REGION Network 63: Reset CMS
   // Reset Axis when the unit is in the resetting state.
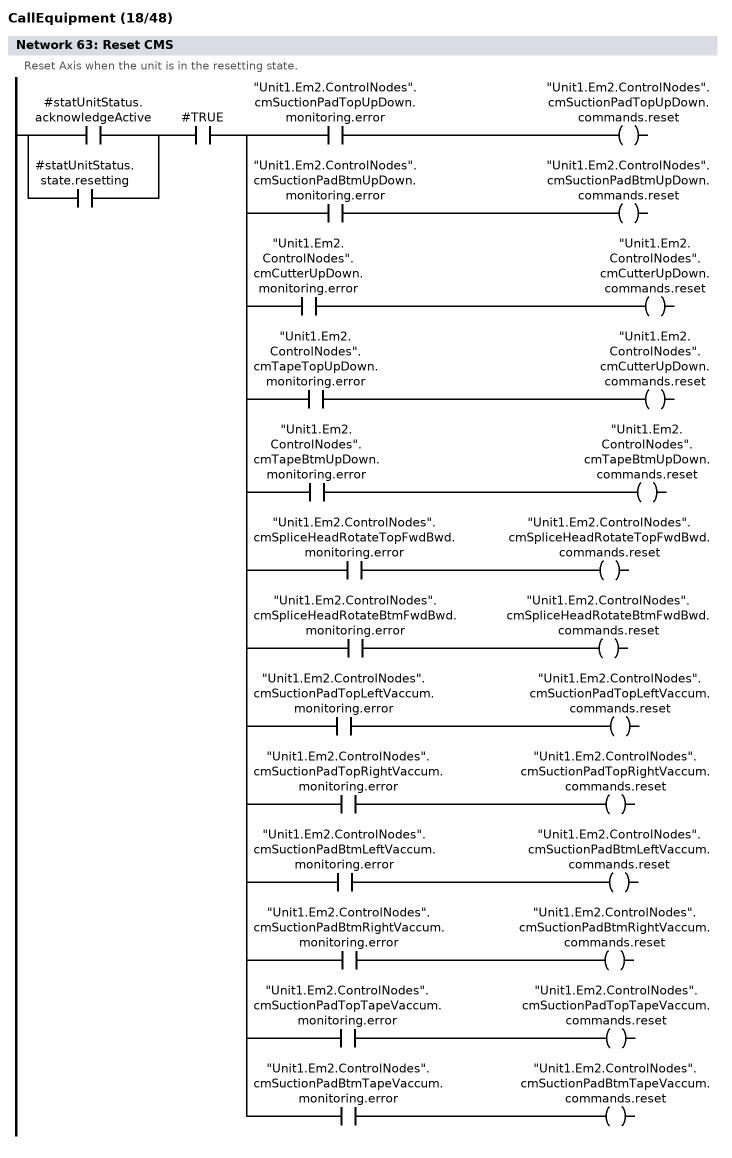
   RUNG wire#powerrail
      Contact( #statUnitStatus.acknowledgeActive )
      wire#w1
      Contact( #TRUE )
      wire#w2
      Contact( "Unit1.Em2.ControlNodes".cmSuctionPadTopUpDown.monitoring.error )
      Coil( "Unit1.Em2.ControlNodes".cmSuctionPadTopUpDown.commands.reset )
   END_RUNG
   RUNG wire#powerrail
      Contact( #statUnitStatus.state.resetting )
   END_RUNG wire#w1
   RUNG wire#w2
      Contact( "Unit1.Em2.ControlNodes".cmSuctionPadBtmUpDown.monitoring.error )
      Coil( "Unit1.Em2.ControlNodes".cmSuctionPadBtmUpDown.commands.reset )
   END_RUNG
   RUNG wire#w2
      Contact( "Unit1.Em2.ControlNodes".cmCutterUpDown.monitoring.error )
      Coil( "Unit1.Em2.ControlNodes".cmCutterUpDown.commands.reset )
   END_RUNG
   RUNG wire#w2
      Contact( "Unit1.Em2.ControlNodes".cmTapeTopUpDown.monitoring.error )
      Coil( "Unit1.Em2.ControlNodes".cmCutterUpDown.commands.reset )
   END_RUNG
   RUNG wire#w2
      Contact( "Unit1.Em2.ControlNodes".cmTapeBtmUpDown.monitoring.error )
      Coil( "Unit1.Em2.ControlNodes".cmTapeBtmUpDown.commands.reset )
   END_RUNG
   RUNG wire#w2
      Contact( "Unit1.Em2.ControlNodes".cmSpliceHeadRotateTopFwdBwd.monitoring.error )
      Coil( "Unit1.Em2.ControlNodes".cmSpliceHeadRotateTopFwdBwd.commands.reset )
   END_RUNG
   RUNG wire#w2
      Contact( "Unit1.Em2.ControlNodes".cmSpliceHeadRotateBtmFwdBwd.monitoring.error )
      Coil( "Unit1.Em2.ControlNodes".cmSpliceHeadRotateBtmFwdBwd.commands.reset )
   END_RUNG
   RUNG wire#w2
      Contact( "Unit1.Em2.ControlNodes".cmSuctionPadTopLeftVaccum.monitoring.error )
      Coil( "Unit1.Em2.ControlNodes".cmSuctionPadTopLeftVaccum.commands.reset )
   END_RUNG
   RUNG wire#w2
      Contact( "Unit1.Em2.ControlNodes".cmSuctionPadTopRightVaccum.monitoring.error )
      Coil( "Unit1.Em2.ControlNodes".cmSuctionPadTopRightVaccum.commands.reset )
   END_RUNG
   RUNG wire#w2
      Contact( "Unit1.Em2.ControlNodes".cmSuctionPadBtmLeftVaccum.monitoring.error )
      Coil( "Unit1.Em2.ControlNodes".cmSuctionPadBtmLeftVaccum.commands.reset )
   END_RUNG
   RUNG wire#w2
      Contact( "Unit1.Em2.ControlNodes".cmSuctionPadBtmRightVaccum.monitoring.error )
      Coil( "Unit1.Em2.ControlNodes".cmSuctionPadBtmRightVaccum.commands.reset )
   END_RUNG
   RUNG wire#w2
      Contact( "Unit1.Em2.ControlNodes".cmSuctionPadTopTapeVaccum.monitoring.error )
      Coil( "Unit1.Em2.ControlNodes".cmSuctionPadTopTapeVaccum.commands.reset )
   END_RUNG
   RUNG wire#w2
      Contact( "Unit1.Em2.ControlNodes".cmSuctionPadBtmTapeVaccum.monitoring.error )
      Coil( "Unit1.Em2.ControlNodes".cmSuctionPadBtmTapeVaccum.commands.reset )
   END_RUNG
   // the same network as SCL:
   #_w1 := (#statUnitStatus.acknowledgeActive OR #statUnitStatus.state.resetting) AND #TRUE;
   "Unit1.Em2.ControlNodes".cmSuctionPadTopUpDown.commands.reset := #_w1 AND "Unit1.Em2.ControlNodes".cmSuctionPadTopUpDown.monitoring.error;
   "Unit1.Em2.ControlNodes".cmSuctionPadBtmUpDown.commands.reset := #_w1 AND "Unit1.Em2.ControlNodes".cmSuctionPadBtmUpDown.monitoring.error;
   "Unit1.Em2.ControlNodes".cmCutterUpDown.commands.reset := #_w1 AND "Unit1.Em2.ControlNodes".cmCutterUpDown.monitoring.error;
   "Unit1.Em2.ControlNodes".cmCutterUpDown.commands.reset := #_w1 AND "Unit1.Em2.ControlNodes".cmTapeTopUpDown.monitoring.error;
   "Unit1.Em2.ControlNodes".cmTapeBtmUpDown.commands.reset := #_w1 AND "Unit1.Em2.ControlNodes".cmTapeBtmUpDown.monitoring.error;
   "Unit1.Em2.ControlNodes".cmSpliceHeadRotateTopFwdBwd.commands.reset := #_w1 AND "Unit1.Em2.ControlNodes".cmSpliceHeadRotateTopFwdBwd.monitoring.error;
   "Unit1.Em2.ControlNodes".cmSpliceHeadRotateBtmFwdBwd.commands.reset := #_w1 AND "Unit1.Em2.ControlNodes".cmSpliceHeadRotateBtmFwdBwd.monitoring.error;
   "Unit1.Em2.ControlNodes".cmSuctionPadTopLeftVaccum.commands.reset := #_w1 AND "Unit1.Em2.ControlNodes".cmSuctionPadTopLeftVaccum.monitoring.error;
   "Unit1.Em2.ControlNodes".cmSuctionPadTopRightVaccum.commands.reset := #_w1 AND "Unit1.Em2.ControlNodes".cmSuctionPadTopRightVaccum.monitoring.error;
   "Unit1.Em2.ControlNodes".cmSuctionPadBtmLeftVaccum.commands.reset := #_w1 AND "Unit1.Em2.ControlNodes".cmSuctionPadBtmLeftVaccum.monitoring.error;
   "Unit1.Em2.ControlNodes".cmSuctionPadBtmRightVaccum.commands.reset := #_w1 AND "Unit1.Em2.ControlNodes".cmSuctionPadBtmRightVaccum.monitoring.error;
   "Unit1.Em2.ControlNodes".cmSuctionPadTopTapeVaccum.commands.reset := #_w1 AND "Unit1.Em2.ControlNodes".cmSuctionPadTopTapeVaccum.monitoring.error;
   "Unit1.Em2.ControlNodes".cmSuctionPadBtmTapeVaccum.commands.reset := #_w1 AND "Unit1.Em2.ControlNodes".cmSuctionPadBtmTapeVaccum.monitoring.error;
END_REGION

REGION Network 65: cmSuctionPadTopUpDown Interlock
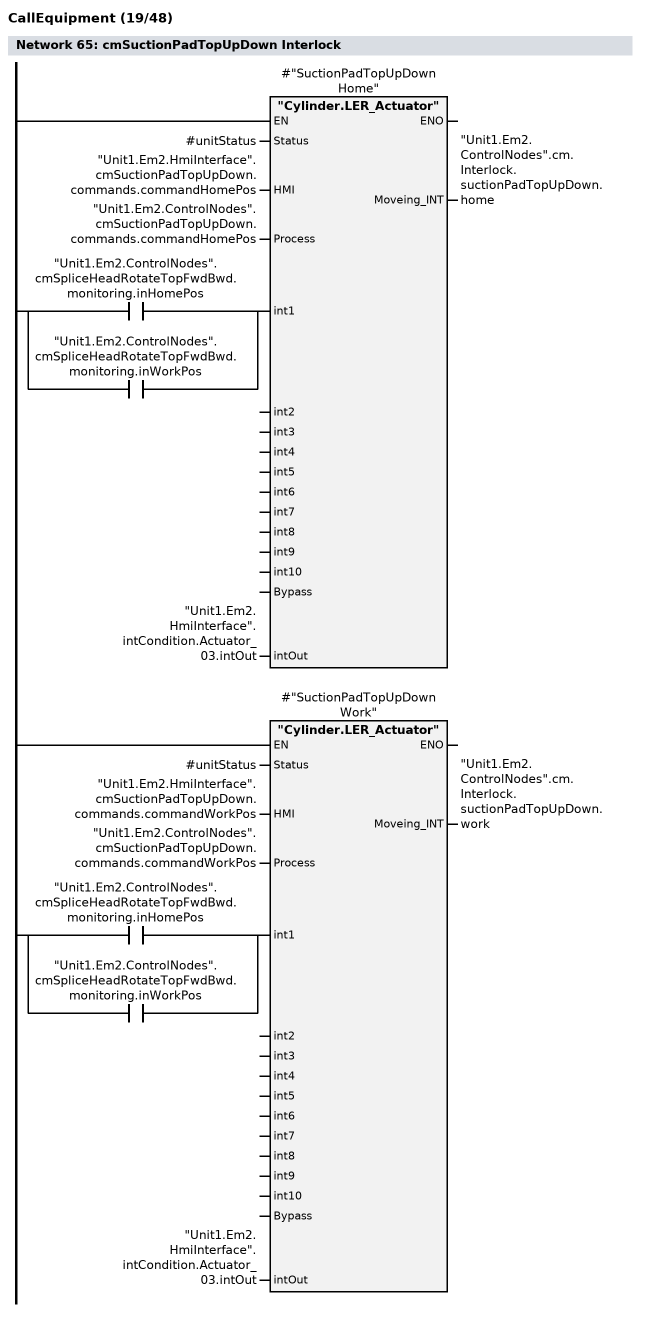
   RUNG wire#powerrail
      #"SuctionPadTopUpDown Home"(int1 := wire#w1, Status := #unitStatus, HMI := "Unit1.Em2.HmiInterface".cmSuctionPadTopUpDown.commands.commandHomePos, Process := "Unit1.Em2.ControlNodes".cmSuctionPadTopUpDown.commands.commandHomePos, int2 :=, int3 :=, int4 :=, int5 :=, int6 :=, int7 :=, int8 :=, int9 :=, int10 :=, Bypass :=, intOut := "Unit1.Em2.HmiInterface".intCondition.Actuator_03.intOut, Moveing_INT => "Unit1.Em2.ControlNodes".cm.Interlock.suctionPadTopUpDown.home)
   END_RUNG
   RUNG wire#powerrail
      Contact( "Unit1.Em2.ControlNodes".cmSpliceHeadRotateTopFwdBwd.monitoring.inHomePos )
   END_RUNG wire#w1
   RUNG wire#powerrail
      Contact( "Unit1.Em2.ControlNodes".cmSpliceHeadRotateTopFwdBwd.monitoring.inWorkPos )
   END_RUNG wire#w1
   RUNG wire#powerrail
      #"SuctionPadTopUpDown Work"(int1 := wire#w2, Status := #unitStatus, HMI := "Unit1.Em2.HmiInterface".cmSuctionPadTopUpDown.commands.commandWorkPos, Process := "Unit1.Em2.ControlNodes".cmSuctionPadTopUpDown.commands.commandWorkPos, int2 :=, int3 :=, int4 :=, int5 :=, int6 :=, int7 :=, int8 :=, int9 :=, int10 :=, Bypass :=, intOut := "Unit1.Em2.HmiInterface".intCondition.Actuator_03.intOut, Moveing_INT => "Unit1.Em2.ControlNodes".cm.Interlock.suctionPadTopUpDown.work)
   END_RUNG
   RUNG wire#powerrail
      Contact( "Unit1.Em2.ControlNodes".cmSpliceHeadRotateTopFwdBwd.monitoring.inHomePos )
   END_RUNG wire#w2
   RUNG wire#powerrail
      Contact( "Unit1.Em2.ControlNodes".cmSpliceHeadRotateTopFwdBwd.monitoring.inWorkPos )
   END_RUNG wire#w2
   // the same network as SCL:
   #"SuctionPadTopUpDown Home"(Status := #unitStatus,   // "Cylinder.LER_Actuator"
                           HMI := "Unit1.Em2.HmiInterface".cmSuctionPadTopUpDown.commands.commandHomePos,
                           Process := "Unit1.Em2.ControlNodes".cmSuctionPadTopUpDown.commands.commandHomePos,
                           int1 := "Unit1.Em2.ControlNodes".cmSpliceHeadRotateTopFwdBwd.monitoring.inHomePos OR "Unit1.Em2.ControlNodes".cmSpliceHeadRotateTopFwdBwd.monitoring.inWorkPos,
                           intOut := "Unit1.Em2.HmiInterface".intCondition.Actuator_03.intOut,
                           Moveing_INT => "Unit1.Em2.ControlNodes".cm.Interlock.suctionPadTopUpDown.home);
   #"SuctionPadTopUpDown Work"(Status := #unitStatus,   // "Cylinder.LER_Actuator"
                           HMI := "Unit1.Em2.HmiInterface".cmSuctionPadTopUpDown.commands.commandWorkPos,
                           Process := "Unit1.Em2.ControlNodes".cmSuctionPadTopUpDown.commands.commandWorkPos,
                           int1 := "Unit1.Em2.ControlNodes".cmSpliceHeadRotateTopFwdBwd.monitoring.inHomePos OR "Unit1.Em2.ControlNodes".cmSpliceHeadRotateTopFwdBwd.monitoring.inWorkPos,
                           intOut := "Unit1.Em2.HmiInterface".intCondition.Actuator_03.intOut,
                           Moveing_INT => "Unit1.Em2.ControlNodes".cm.Interlock.suctionPadTopUpDown.work);
END_REGION

REGION Network 66: cmSuctionPadTopUpDown Commands
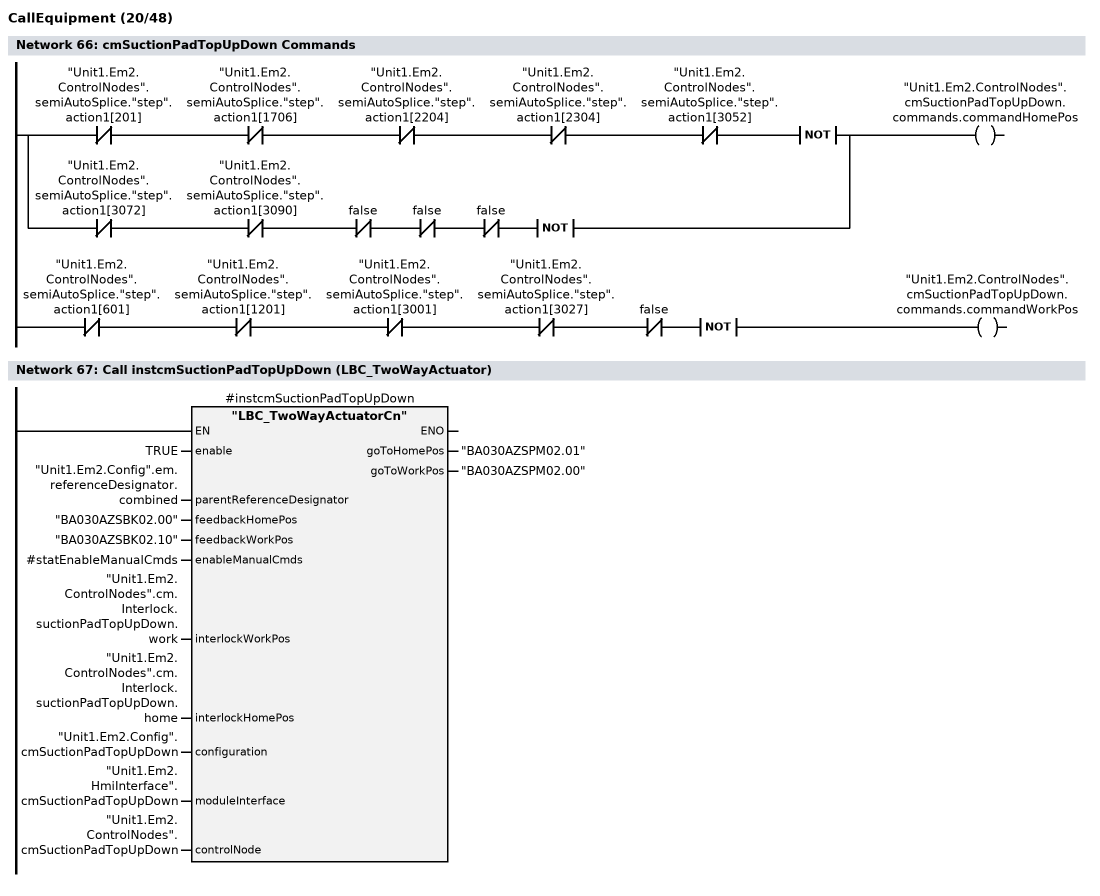
   RUNG wire#powerrail
      I_Contact( "Unit1.Em2.ControlNodes".semiAutoSplice."step".action1[201] )
      I_Contact( "Unit1.Em2.ControlNodes".semiAutoSplice."step".action1[1706] )
      I_Contact( "Unit1.Em2.ControlNodes".semiAutoSplice."step".action1[2204] )
      I_Contact( "Unit1.Em2.ControlNodes".semiAutoSplice."step".action1[2304] )
      I_Contact( "Unit1.Em2.ControlNodes".semiAutoSplice."step".action1[3052] )
      Not()
      wire#w1
      Coil( "Unit1.Em2.ControlNodes".cmSuctionPadTopUpDown.commands.commandHomePos )
   END_RUNG
   RUNG wire#powerrail
      I_Contact( "Unit1.Em2.ControlNodes".semiAutoSplice."step".action1[3072] )
      I_Contact( "Unit1.Em2.ControlNodes".semiAutoSplice."step".action1[3090] )
      I_Contact( false )
      I_Contact( false )
      I_Contact( false )
      Not()
   END_RUNG wire#w1
   RUNG wire#powerrail
      I_Contact( "Unit1.Em2.ControlNodes".semiAutoSplice."step".action1[601] )
      I_Contact( "Unit1.Em2.ControlNodes".semiAutoSplice."step".action1[1201] )
      I_Contact( "Unit1.Em2.ControlNodes".semiAutoSplice."step".action1[3001] )
      I_Contact( "Unit1.Em2.ControlNodes".semiAutoSplice."step".action1[3027] )
      I_Contact( false )
      Not()
      Coil( "Unit1.Em2.ControlNodes".cmSuctionPadTopUpDown.commands.commandWorkPos )
   END_RUNG
   // the same network as SCL:
   "Unit1.Em2.ControlNodes".cmSuctionPadTopUpDown.commands.commandHomePos := NOT (NOT "Unit1.Em2.ControlNodes".semiAutoSplice."step".action1[201] AND NOT "Unit1.Em2.ControlNodes".semiAutoSplice."step".action1[1706] AND NOT "Unit1.Em2.ControlNodes".semiAutoSplice."step".action1[2204] AND NOT "Unit1.Em2.ControlNodes".semiAutoSplice."step".action1[2304] AND NOT "Unit1.Em2.ControlNodes".semiAutoSplice."step".action1[3052]) OR NOT (NOT "Unit1.Em2.ControlNodes".semiAutoSplice."step".action1[3072] AND NOT "Unit1.Em2.ControlNodes".semiAutoSplice."step".action1[3090] AND NOT false AND NOT false AND NOT false);
   "Unit1.Em2.ControlNodes".cmSuctionPadTopUpDown.commands.commandWorkPos := NOT (NOT "Unit1.Em2.ControlNodes".semiAutoSplice."step".action1[601] AND NOT "Unit1.Em2.ControlNodes".semiAutoSplice."step".action1[1201] AND NOT "Unit1.Em2.ControlNodes".semiAutoSplice."step".action1[3001] AND NOT "Unit1.Em2.ControlNodes".semiAutoSplice."step".action1[3027] AND NOT false);
END_REGION

REGION Network 67: Call instcmSuctionPadTopUpDown (LBC_TwoWayActuator)
   RUNG wire#powerrail
      #instcmSuctionPadTopUpDown(enable := TRUE, parentReferenceDesignator := "Unit1.Em2.Config".em.referenceDesignator.combined, feedbackHomePos := "BA030AZSBK02.00", feedbackWorkPos := "BA030AZSBK02.10", enableManualCmds := #statEnableManualCmds, interlockWorkPos := "Unit1.Em2.ControlNodes".cm.Interlock.suctionPadTopUpDown.work, interlockHomePos := "Unit1.Em2.ControlNodes".cm.Interlock.suctionPadTopUpDown.home, configuration := "Unit1.Em2.Config".cmSuctionPadTopUpDown, moduleInterface := "Unit1.Em2.HmiInterface".cmSuctionPadTopUpDown, controlNode := "Unit1.Em2.ControlNodes".cmSuctionPadTopUpDown, goToHomePos => "BA030AZSPM02.01", goToWorkPos => "BA030AZSPM02.00")
   END_RUNG
   // the same network as SCL:
   #instcmSuctionPadTopUpDown(enable := TRUE,   // "LBC_TwoWayActuatorCn"
                           parentReferenceDesignator := "Unit1.Em2.Config".em.referenceDesignator.combined,
                           feedbackHomePos := "BA030AZSBK02.00",
                           feedbackWorkPos := "BA030AZSBK02.10",
                           enableManualCmds := #statEnableManualCmds,
                           interlockWorkPos := "Unit1.Em2.ControlNodes".cm.Interlock.suctionPadTopUpDown.work,
                           interlockHomePos := "Unit1.Em2.ControlNodes".cm.Interlock.suctionPadTopUpDown.home,
                           configuration := "Unit1.Em2.Config".cmSuctionPadTopUpDown,
                           moduleInterface := "Unit1.Em2.HmiInterface".cmSuctionPadTopUpDown,
                           controlNode := "Unit1.Em2.ControlNodes".cmSuctionPadTopUpDown,
                           goToHomePos => "BA030AZSPM02.01",
                           goToWorkPos => "BA030AZSPM02.00");
END_REGION

REGION Network 69: cmSuctionPadBtmUpDown Interlock
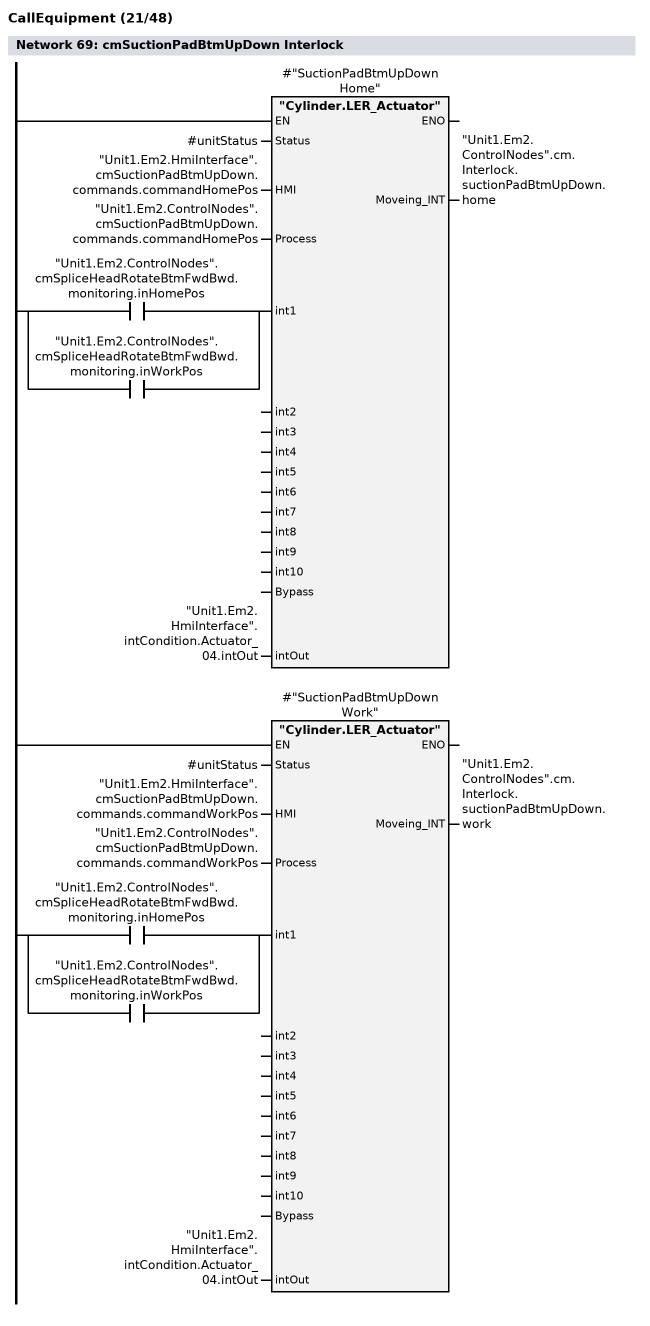
   RUNG wire#powerrail
      #"SuctionPadBtmUpDown Home"(int1 := wire#w1, Status := #unitStatus, HMI := "Unit1.Em2.HmiInterface".cmSuctionPadBtmUpDown.commands.commandHomePos, Process := "Unit1.Em2.ControlNodes".cmSuctionPadBtmUpDown.commands.commandHomePos, int2 :=, int3 :=, int4 :=, int5 :=, int6 :=, int7 :=, int8 :=, int9 :=, int10 :=, Bypass :=, intOut := "Unit1.Em2.HmiInterface".intCondition.Actuator_04.intOut, Moveing_INT => "Unit1.Em2.ControlNodes".cm.Interlock.suctionPadBtmUpDown.home)
   END_RUNG
   RUNG wire#powerrail
      Contact( "Unit1.Em2.ControlNodes".cmSpliceHeadRotateBtmFwdBwd.monitoring.inHomePos )
   END_RUNG wire#w1
   RUNG wire#powerrail
      Contact( "Unit1.Em2.ControlNodes".cmSpliceHeadRotateBtmFwdBwd.monitoring.inWorkPos )
   END_RUNG wire#w1
   RUNG wire#powerrail
      #"SuctionPadBtmUpDown Work"(int1 := wire#w2, Status := #unitStatus, HMI := "Unit1.Em2.HmiInterface".cmSuctionPadBtmUpDown.commands.commandWorkPos, Process := "Unit1.Em2.ControlNodes".cmSuctionPadBtmUpDown.commands.commandWorkPos, int2 :=, int3 :=, int4 :=, int5 :=, int6 :=, int7 :=, int8 :=, int9 :=, int10 :=, Bypass :=, intOut := "Unit1.Em2.HmiInterface".intCondition.Actuator_04.intOut, Moveing_INT => "Unit1.Em2.ControlNodes".cm.Interlock.suctionPadBtmUpDown.work)
   END_RUNG
   RUNG wire#powerrail
      Contact( "Unit1.Em2.ControlNodes".cmSpliceHeadRotateBtmFwdBwd.monitoring.inHomePos )
   END_RUNG wire#w2
   RUNG wire#powerrail
      Contact( "Unit1.Em2.ControlNodes".cmSpliceHeadRotateBtmFwdBwd.monitoring.inWorkPos )
   END_RUNG wire#w2
   // the same network as SCL:
   #"SuctionPadBtmUpDown Home"(Status := #unitStatus,   // "Cylinder.LER_Actuator"
                           HMI := "Unit1.Em2.HmiInterface".cmSuctionPadBtmUpDown.commands.commandHomePos,
                           Process := "Unit1.Em2.ControlNodes".cmSuctionPadBtmUpDown.commands.commandHomePos,
                           int1 := "Unit1.Em2.ControlNodes".cmSpliceHeadRotateBtmFwdBwd.monitoring.inHomePos OR "Unit1.Em2.ControlNodes".cmSpliceHeadRotateBtmFwdBwd.monitoring.inWorkPos,
                           intOut := "Unit1.Em2.HmiInterface".intCondition.Actuator_04.intOut,
                           Moveing_INT => "Unit1.Em2.ControlNodes".cm.Interlock.suctionPadBtmUpDown.home);
   #"SuctionPadBtmUpDown Work"(Status := #unitStatus,   // "Cylinder.LER_Actuator"
                           HMI := "Unit1.Em2.HmiInterface".cmSuctionPadBtmUpDown.commands.commandWorkPos,
                           Process := "Unit1.Em2.ControlNodes".cmSuctionPadBtmUpDown.commands.commandWorkPos,
                           int1 := "Unit1.Em2.ControlNodes".cmSpliceHeadRotateBtmFwdBwd.monitoring.inHomePos OR "Unit1.Em2.ControlNodes".cmSpliceHeadRotateBtmFwdBwd.monitoring.inWorkPos,
                           intOut := "Unit1.Em2.HmiInterface".intCondition.Actuator_04.intOut,
                           Moveing_INT => "Unit1.Em2.ControlNodes".cm.Interlock.suctionPadBtmUpDown.work);
END_REGION

REGION Network 70: cmSuctionPadBtmUpDown Commands
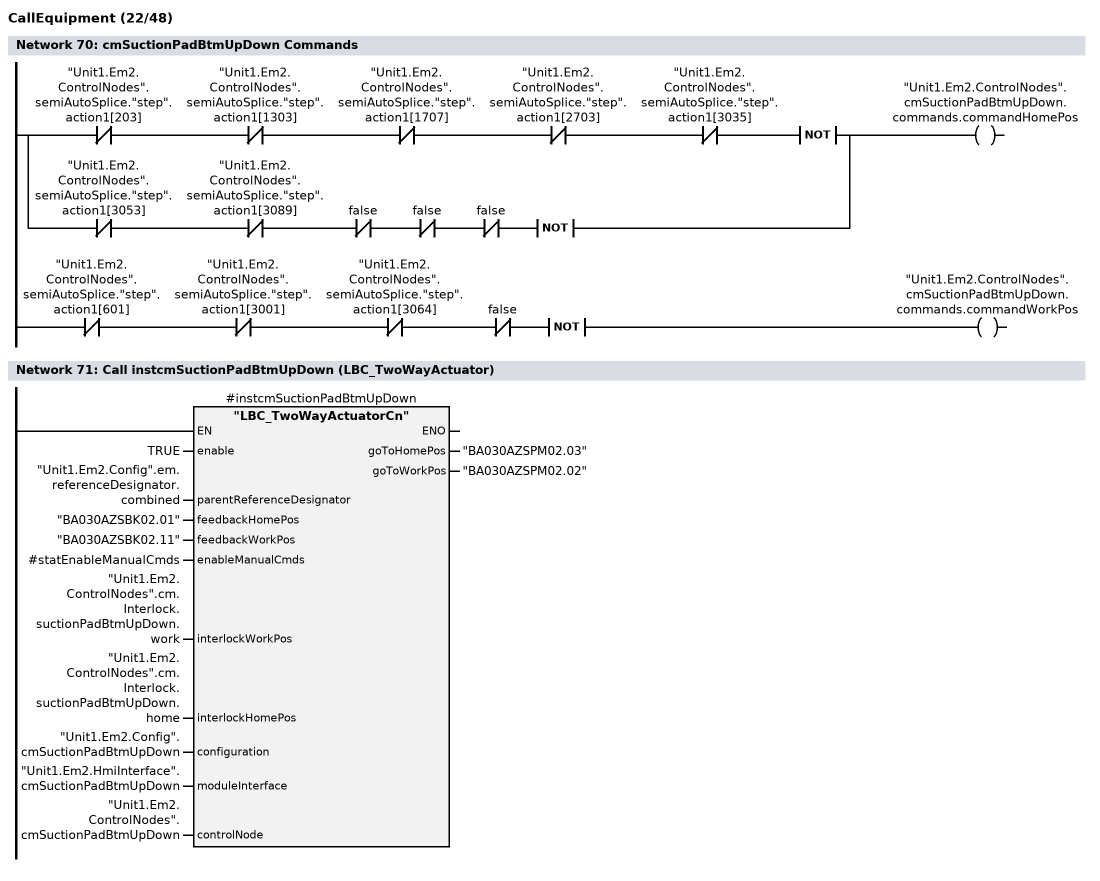
   RUNG wire#powerrail
      I_Contact( "Unit1.Em2.ControlNodes".semiAutoSplice."step".action1[203] )
      I_Contact( "Unit1.Em2.ControlNodes".semiAutoSplice."step".action1[1303] )
      I_Contact( "Unit1.Em2.ControlNodes".semiAutoSplice."step".action1[1707] )
      I_Contact( "Unit1.Em2.ControlNodes".semiAutoSplice."step".action1[2703] )
      I_Contact( "Unit1.Em2.ControlNodes".semiAutoSplice."step".action1[3035] )
      Not()
      wire#w1
      Coil( "Unit1.Em2.ControlNodes".cmSuctionPadBtmUpDown.commands.commandHomePos )
   END_RUNG
   RUNG wire#powerrail
      I_Contact( "Unit1.Em2.ControlNodes".semiAutoSplice."step".action1[3053] )
      I_Contact( "Unit1.Em2.ControlNodes".semiAutoSplice."step".action1[3089] )
      I_Contact( false )
      I_Contact( false )
      I_Contact( false )
      Not()
   END_RUNG wire#w1
   RUNG wire#powerrail
      I_Contact( "Unit1.Em2.ControlNodes".semiAutoSplice."step".action1[601] )
      I_Contact( "Unit1.Em2.ControlNodes".semiAutoSplice."step".action1[3001] )
      I_Contact( "Unit1.Em2.ControlNodes".semiAutoSplice."step".action1[3064] )
      I_Contact( false )
      Not()
      Coil( "Unit1.Em2.ControlNodes".cmSuctionPadBtmUpDown.commands.commandWorkPos )
   END_RUNG
   // the same network as SCL:
   "Unit1.Em2.ControlNodes".cmSuctionPadBtmUpDown.commands.commandHomePos := NOT (NOT "Unit1.Em2.ControlNodes".semiAutoSplice."step".action1[203] AND NOT "Unit1.Em2.ControlNodes".semiAutoSplice."step".action1[1303] AND NOT "Unit1.Em2.ControlNodes".semiAutoSplice."step".action1[1707] AND NOT "Unit1.Em2.ControlNodes".semiAutoSplice."step".action1[2703] AND NOT "Unit1.Em2.ControlNodes".semiAutoSplice."step".action1[3035]) OR NOT (NOT "Unit1.Em2.ControlNodes".semiAutoSplice."step".action1[3053] AND NOT "Unit1.Em2.ControlNodes".semiAutoSplice."step".action1[3089] AND NOT false AND NOT false AND NOT false);
   "Unit1.Em2.ControlNodes".cmSuctionPadBtmUpDown.commands.commandWorkPos := NOT (NOT "Unit1.Em2.ControlNodes".semiAutoSplice."step".action1[601] AND NOT "Unit1.Em2.ControlNodes".semiAutoSplice."step".action1[3001] AND NOT "Unit1.Em2.ControlNodes".semiAutoSplice."step".action1[3064] AND NOT false);
END_REGION

REGION Network 71: Call instcmSuctionPadBtmUpDown (LBC_TwoWayActuator)
   RUNG wire#powerrail
      #instcmSuctionPadBtmUpDown(enable := TRUE, parentReferenceDesignator := "Unit1.Em2.Config".em.referenceDesignator.combined, feedbackHomePos := "BA030AZSBK02.01", feedbackWorkPos := "BA030AZSBK02.11", enableManualCmds := #statEnableManualCmds, interlockWorkPos := "Unit1.Em2.ControlNodes".cm.Interlock.suctionPadBtmUpDown.work, interlockHomePos := "Unit1.Em2.ControlNodes".cm.Interlock.suctionPadBtmUpDown.home, configuration := "Unit1.Em2.Config".cmSuctionPadBtmUpDown, moduleInterface := "Unit1.Em2.HmiInterface".cmSuctionPadBtmUpDown, controlNode := "Unit1.Em2.ControlNodes".cmSuctionPadBtmUpDown, goToHomePos => "BA030AZSPM02.03", goToWorkPos => "BA030AZSPM02.02")
   END_RUNG
   // the same network as SCL:
   #instcmSuctionPadBtmUpDown(enable := TRUE,   // "LBC_TwoWayActuatorCn"
                           parentReferenceDesignator := "Unit1.Em2.Config".em.referenceDesignator.combined,
                           feedbackHomePos := "BA030AZSBK02.01",
                           feedbackWorkPos := "BA030AZSBK02.11",
                           enableManualCmds := #statEnableManualCmds,
                           interlockWorkPos := "Unit1.Em2.ControlNodes".cm.Interlock.suctionPadBtmUpDown.work,
                           interlockHomePos := "Unit1.Em2.ControlNodes".cm.Interlock.suctionPadBtmUpDown.home,
                           configuration := "Unit1.Em2.Config".cmSuctionPadBtmUpDown,
                           moduleInterface := "Unit1.Em2.HmiInterface".cmSuctionPadBtmUpDown,
                           controlNode := "Unit1.Em2.ControlNodes".cmSuctionPadBtmUpDown,
                           goToHomePos => "BA030AZSPM02.03",
                           goToWorkPos => "BA030AZSPM02.02");
END_REGION

REGION Network 73: cmCutterUpDown Interlock
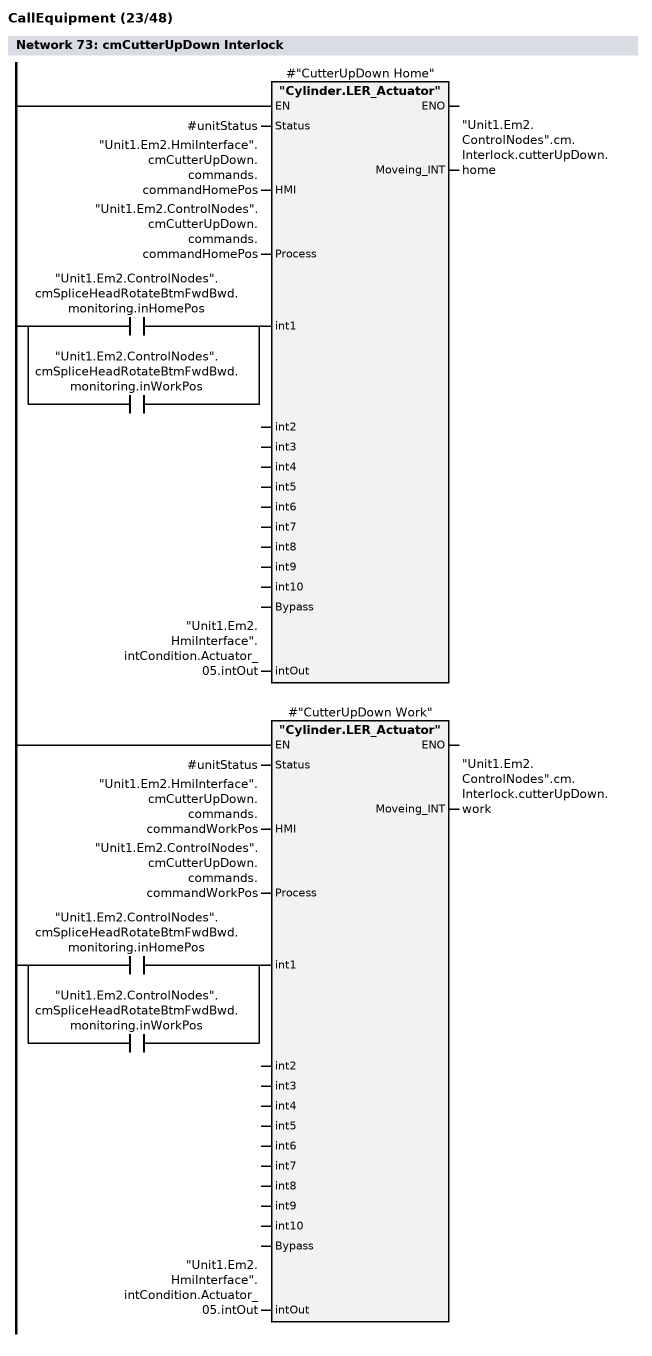
   RUNG wire#powerrail
      #"CutterUpDown Home"(int1 := wire#w1, Status := #unitStatus, HMI := "Unit1.Em2.HmiInterface".cmCutterUpDown.commands.commandHomePos, Process := "Unit1.Em2.ControlNodes".cmCutterUpDown.commands.commandHomePos, int2 :=, int3 :=, int4 :=, int5 :=, int6 :=, int7 :=, int8 :=, int9 :=, int10 :=, Bypass :=, intOut := "Unit1.Em2.HmiInterface".intCondition.Actuator_05.intOut, Moveing_INT => "Unit1.Em2.ControlNodes".cm.Interlock.cutterUpDown.home)
   END_RUNG
   RUNG wire#powerrail
      Contact( "Unit1.Em2.ControlNodes".cmSpliceHeadRotateBtmFwdBwd.monitoring.inHomePos )
   END_RUNG wire#w1
   RUNG wire#powerrail
      Contact( "Unit1.Em2.ControlNodes".cmSpliceHeadRotateBtmFwdBwd.monitoring.inWorkPos )
   END_RUNG wire#w1
   RUNG wire#powerrail
      #"CutterUpDown Work"(int1 := wire#w2, Status := #unitStatus, HMI := "Unit1.Em2.HmiInterface".cmCutterUpDown.commands.commandWorkPos, Process := "Unit1.Em2.ControlNodes".cmCutterUpDown.commands.commandWorkPos, int2 :=, int3 :=, int4 :=, int5 :=, int6 :=, int7 :=, int8 :=, int9 :=, int10 :=, Bypass :=, intOut := "Unit1.Em2.HmiInterface".intCondition.Actuator_05.intOut, Moveing_INT => "Unit1.Em2.ControlNodes".cm.Interlock.cutterUpDown.work)
   END_RUNG
   RUNG wire#powerrail
      Contact( "Unit1.Em2.ControlNodes".cmSpliceHeadRotateBtmFwdBwd.monitoring.inHomePos )
   END_RUNG wire#w2
   RUNG wire#powerrail
      Contact( "Unit1.Em2.ControlNodes".cmSpliceHeadRotateBtmFwdBwd.monitoring.inWorkPos )
   END_RUNG wire#w2
   // the same network as SCL:
   #"CutterUpDown Home"(Status := #unitStatus,   // "Cylinder.LER_Actuator"
                        HMI := "Unit1.Em2.HmiInterface".cmCutterUpDown.commands.commandHomePos,
                        Process := "Unit1.Em2.ControlNodes".cmCutterUpDown.commands.commandHomePos,
                        int1 := "Unit1.Em2.ControlNodes".cmSpliceHeadRotateBtmFwdBwd.monitoring.inHomePos OR "Unit1.Em2.ControlNodes".cmSpliceHeadRotateBtmFwdBwd.monitoring.inWorkPos,
                        intOut := "Unit1.Em2.HmiInterface".intCondition.Actuator_05.intOut,
                        Moveing_INT => "Unit1.Em2.ControlNodes".cm.Interlock.cutterUpDown.home);
   #"CutterUpDown Work"(Status := #unitStatus,   // "Cylinder.LER_Actuator"
                        HMI := "Unit1.Em2.HmiInterface".cmCutterUpDown.commands.commandWorkPos,
                        Process := "Unit1.Em2.ControlNodes".cmCutterUpDown.commands.commandWorkPos,
                        int1 := "Unit1.Em2.ControlNodes".cmSpliceHeadRotateBtmFwdBwd.monitoring.inHomePos OR "Unit1.Em2.ControlNodes".cmSpliceHeadRotateBtmFwdBwd.monitoring.inWorkPos,
                        intOut := "Unit1.Em2.HmiInterface".intCondition.Actuator_05.intOut,
                        Moveing_INT => "Unit1.Em2.ControlNodes".cm.Interlock.cutterUpDown.work);
END_REGION

REGION Network 74: cmCutterUpDown Commands
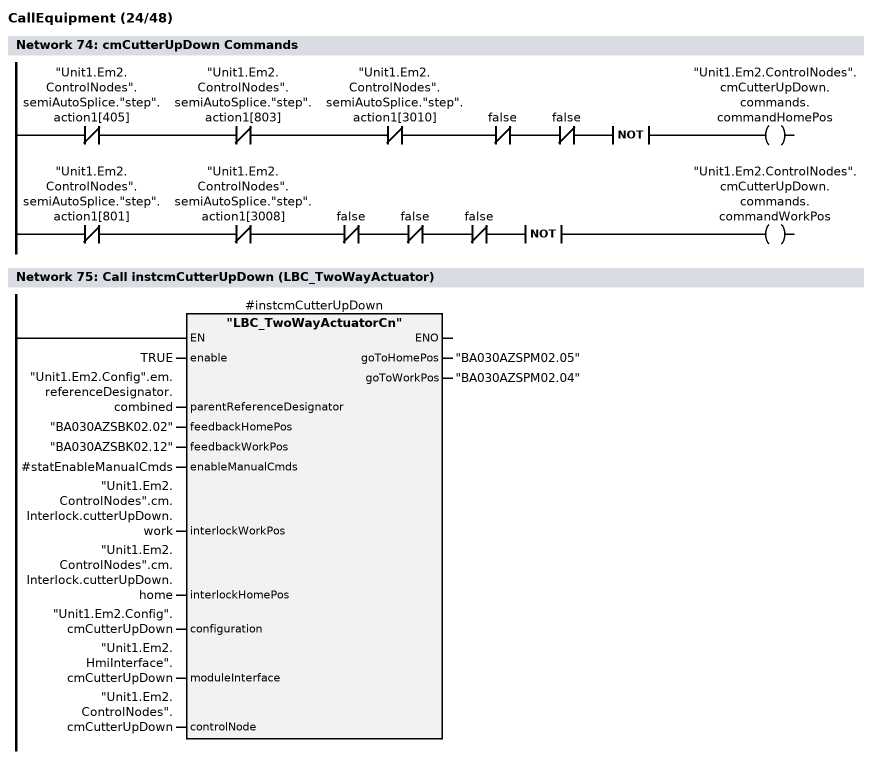
   RUNG wire#powerrail
      I_Contact( "Unit1.Em2.ControlNodes".semiAutoSplice."step".action1[405] )
      I_Contact( "Unit1.Em2.ControlNodes".semiAutoSplice."step".action1[803] )
      I_Contact( "Unit1.Em2.ControlNodes".semiAutoSplice."step".action1[3010] )
      I_Contact( false )
      I_Contact( false )
      Not()
      Coil( "Unit1.Em2.ControlNodes".cmCutterUpDown.commands.commandHomePos )
   END_RUNG
   RUNG wire#powerrail
      I_Contact( "Unit1.Em2.ControlNodes".semiAutoSplice."step".action1[801] )
      I_Contact( "Unit1.Em2.ControlNodes".semiAutoSplice."step".action1[3008] )
      I_Contact( false )
      I_Contact( false )
      I_Contact( false )
      Not()
      Coil( "Unit1.Em2.ControlNodes".cmCutterUpDown.commands.commandWorkPos )
   END_RUNG
   // the same network as SCL:
   "Unit1.Em2.ControlNodes".cmCutterUpDown.commands.commandHomePos := NOT (NOT "Unit1.Em2.ControlNodes".semiAutoSplice."step".action1[405] AND NOT "Unit1.Em2.ControlNodes".semiAutoSplice."step".action1[803] AND NOT "Unit1.Em2.ControlNodes".semiAutoSplice."step".action1[3010] AND NOT false AND NOT false);
   "Unit1.Em2.ControlNodes".cmCutterUpDown.commands.commandWorkPos := NOT (NOT "Unit1.Em2.ControlNodes".semiAutoSplice."step".action1[801] AND NOT "Unit1.Em2.ControlNodes".semiAutoSplice."step".action1[3008] AND NOT false AND NOT false AND NOT false);
END_REGION

REGION Network 75: Call instcmCutterUpDown (LBC_TwoWayActuator)
   RUNG wire#powerrail
      #instcmCutterUpDown(enable := TRUE, parentReferenceDesignator := "Unit1.Em2.Config".em.referenceDesignator.combined, feedbackHomePos := "BA030AZSBK02.02", feedbackWorkPos := "BA030AZSBK02.12", enableManualCmds := #statEnableManualCmds, interlockWorkPos := "Unit1.Em2.ControlNodes".cm.Interlock.cutterUpDown.work, interlockHomePos := "Unit1.Em2.ControlNodes".cm.Interlock.cutterUpDown.home, configuration := "Unit1.Em2.Config".cmCutterUpDown, moduleInterface := "Unit1.Em2.HmiInterface".cmCutterUpDown, controlNode := "Unit1.Em2.ControlNodes".cmCutterUpDown, goToHomePos => "BA030AZSPM02.05", goToWorkPos => "BA030AZSPM02.04")
   END_RUNG
   // the same network as SCL:
   #instcmCutterUpDown(enable := TRUE,   // "LBC_TwoWayActuatorCn"
                       parentReferenceDesignator := "Unit1.Em2.Config".em.referenceDesignator.combined,
                       feedbackHomePos := "BA030AZSBK02.02",
                       feedbackWorkPos := "BA030AZSBK02.12",
                       enableManualCmds := #statEnableManualCmds,
                       interlockWorkPos := "Unit1.Em2.ControlNodes".cm.Interlock.cutterUpDown.work,
                       interlockHomePos := "Unit1.Em2.ControlNodes".cm.Interlock.cutterUpDown.home,
                       configuration := "Unit1.Em2.Config".cmCutterUpDown,
                       moduleInterface := "Unit1.Em2.HmiInterface".cmCutterUpDown,
                       controlNode := "Unit1.Em2.ControlNodes".cmCutterUpDown,
                       goToHomePos => "BA030AZSPM02.05",
                       goToWorkPos => "BA030AZSPM02.04");
END_REGION

REGION Network 77: cmTapeTopUpDown Interlock
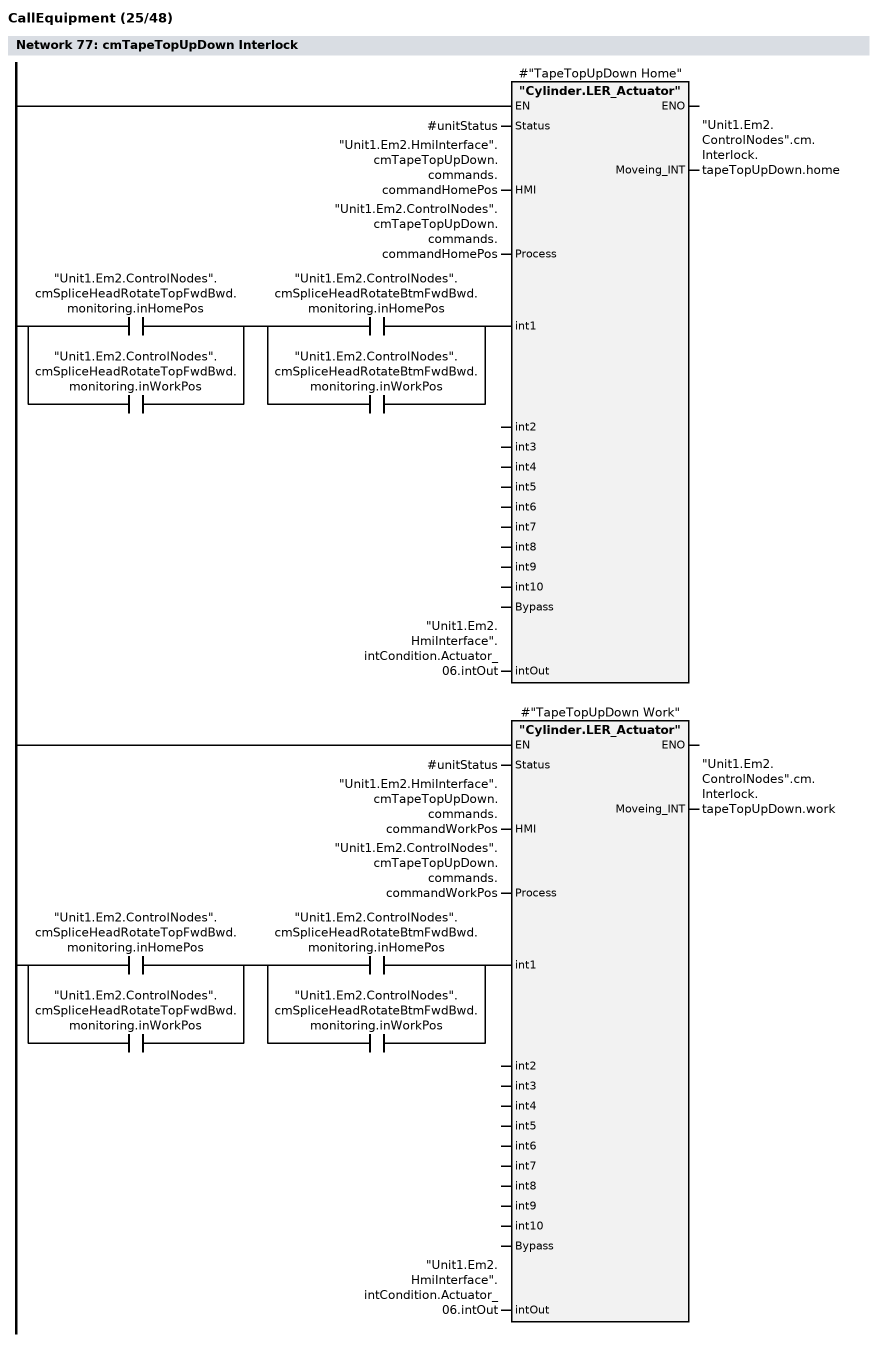
   RUNG wire#powerrail
      #"TapeTopUpDown Home"(int1 := wire#w2, Status := #unitStatus, HMI := "Unit1.Em2.HmiInterface".cmTapeTopUpDown.commands.commandHomePos, Process := "Unit1.Em2.ControlNodes".cmTapeTopUpDown.commands.commandHomePos, int2 :=, int3 :=, int4 :=, int5 :=, int6 :=, int7 :=, int8 :=, int9 :=, int10 :=, Bypass :=, intOut := "Unit1.Em2.HmiInterface".intCondition.Actuator_06.intOut, Moveing_INT => "Unit1.Em2.ControlNodes".cm.Interlock.tapeTopUpDown.home)
   END_RUNG
   RUNG wire#powerrail
      Contact( "Unit1.Em2.ControlNodes".cmSpliceHeadRotateTopFwdBwd.monitoring.inHomePos )
      wire#w1
      Contact( "Unit1.Em2.ControlNodes".cmSpliceHeadRotateBtmFwdBwd.monitoring.inHomePos )
   END_RUNG wire#w2
   RUNG wire#powerrail
      Contact( "Unit1.Em2.ControlNodes".cmSpliceHeadRotateTopFwdBwd.monitoring.inWorkPos )
   END_RUNG wire#w1
   RUNG wire#w1
      Contact( "Unit1.Em2.ControlNodes".cmSpliceHeadRotateBtmFwdBwd.monitoring.inWorkPos )
   END_RUNG wire#w2
   RUNG wire#powerrail
      #"TapeTopUpDown Work"(int1 := wire#w4, Status := #unitStatus, HMI := "Unit1.Em2.HmiInterface".cmTapeTopUpDown.commands.commandWorkPos, Process := "Unit1.Em2.ControlNodes".cmTapeTopUpDown.commands.commandWorkPos, int2 :=, int3 :=, int4 :=, int5 :=, int6 :=, int7 :=, int8 :=, int9 :=, int10 :=, Bypass :=, intOut := "Unit1.Em2.HmiInterface".intCondition.Actuator_06.intOut, Moveing_INT => "Unit1.Em2.ControlNodes".cm.Interlock.tapeTopUpDown.work)
   END_RUNG
   RUNG wire#powerrail
      Contact( "Unit1.Em2.ControlNodes".cmSpliceHeadRotateTopFwdBwd.monitoring.inHomePos )
      wire#w3
      Contact( "Unit1.Em2.ControlNodes".cmSpliceHeadRotateBtmFwdBwd.monitoring.inHomePos )
   END_RUNG wire#w4
   RUNG wire#powerrail
      Contact( "Unit1.Em2.ControlNodes".cmSpliceHeadRotateTopFwdBwd.monitoring.inWorkPos )
   END_RUNG wire#w3
   RUNG wire#w3
      Contact( "Unit1.Em2.ControlNodes".cmSpliceHeadRotateBtmFwdBwd.monitoring.inWorkPos )
   END_RUNG wire#w4
   // the same network as SCL:
   #"TapeTopUpDown Home"(Status := #unitStatus,   // "Cylinder.LER_Actuator"
                         HMI := "Unit1.Em2.HmiInterface".cmTapeTopUpDown.commands.commandHomePos,
                         Process := "Unit1.Em2.ControlNodes".cmTapeTopUpDown.commands.commandHomePos,
                         int1 := ("Unit1.Em2.ControlNodes".cmSpliceHeadRotateTopFwdBwd.monitoring.inHomePos OR "Unit1.Em2.ControlNodes".cmSpliceHeadRotateTopFwdBwd.monitoring.inWorkPos) AND ("Unit1.Em2.ControlNodes".cmSpliceHeadRotateBtmFwdBwd.monitoring.inHomePos OR "Unit1.Em2.ControlNodes".cmSpliceHeadRotateBtmFwdBwd.monitoring.inWorkPos),
                         intOut := "Unit1.Em2.HmiInterface".intCondition.Actuator_06.intOut,
                         Moveing_INT => "Unit1.Em2.ControlNodes".cm.Interlock.tapeTopUpDown.home);
   #"TapeTopUpDown Work"(Status := #unitStatus,   // "Cylinder.LER_Actuator"
                         HMI := "Unit1.Em2.HmiInterface".cmTapeTopUpDown.commands.commandWorkPos,
                         Process := "Unit1.Em2.ControlNodes".cmTapeTopUpDown.commands.commandWorkPos,
                         int1 := ("Unit1.Em2.ControlNodes".cmSpliceHeadRotateTopFwdBwd.monitoring.inHomePos OR "Unit1.Em2.ControlNodes".cmSpliceHeadRotateTopFwdBwd.monitoring.inWorkPos) AND ("Unit1.Em2.ControlNodes".cmSpliceHeadRotateBtmFwdBwd.monitoring.inHomePos OR "Unit1.Em2.ControlNodes".cmSpliceHeadRotateBtmFwdBwd.monitoring.inWorkPos),
                         intOut := "Unit1.Em2.HmiInterface".intCondition.Actuator_06.intOut,
                         Moveing_INT => "Unit1.Em2.ControlNodes".cm.Interlock.tapeTopUpDown.work);
END_REGION

REGION Network 78: cmTapeTopUpDown Commands
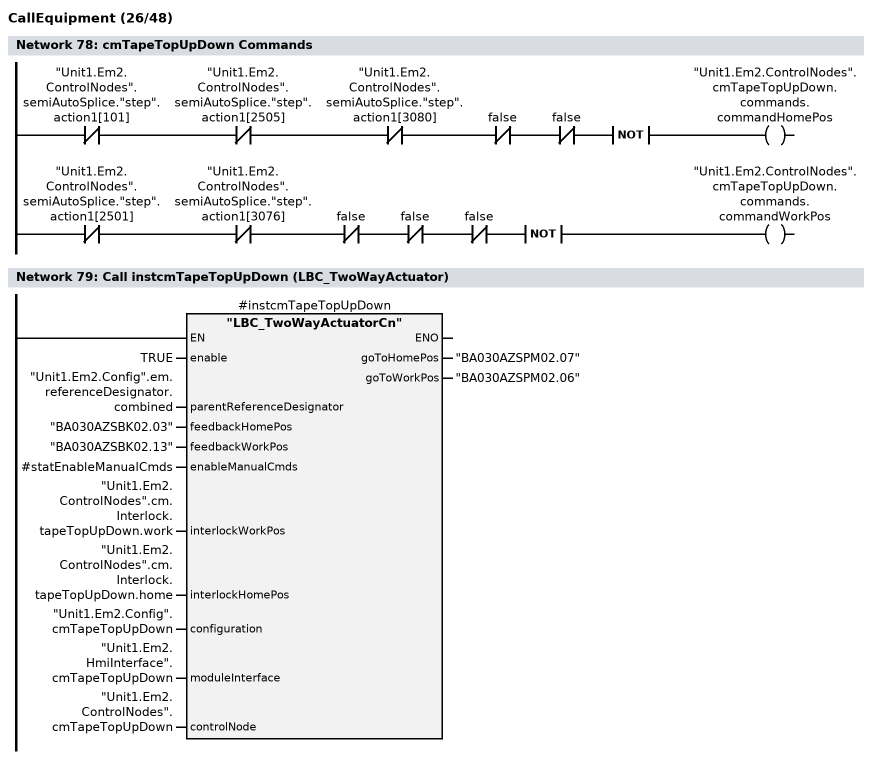
   RUNG wire#powerrail
      I_Contact( "Unit1.Em2.ControlNodes".semiAutoSplice."step".action1[101] )
      I_Contact( "Unit1.Em2.ControlNodes".semiAutoSplice."step".action1[2505] )
      I_Contact( "Unit1.Em2.ControlNodes".semiAutoSplice."step".action1[3080] )
      I_Contact( false )
      I_Contact( false )
      Not()
      Coil( "Unit1.Em2.ControlNodes".cmTapeTopUpDown.commands.commandHomePos )
   END_RUNG
   RUNG wire#powerrail
      I_Contact( "Unit1.Em2.ControlNodes".semiAutoSplice."step".action1[2501] )
      I_Contact( "Unit1.Em2.ControlNodes".semiAutoSplice."step".action1[3076] )
      I_Contact( false )
      I_Contact( false )
      I_Contact( false )
      Not()
      Coil( "Unit1.Em2.ControlNodes".cmTapeTopUpDown.commands.commandWorkPos )
   END_RUNG
   // the same network as SCL:
   "Unit1.Em2.ControlNodes".cmTapeTopUpDown.commands.commandHomePos := NOT (NOT "Unit1.Em2.ControlNodes".semiAutoSplice."step".action1[101] AND NOT "Unit1.Em2.ControlNodes".semiAutoSplice."step".action1[2505] AND NOT "Unit1.Em2.ControlNodes".semiAutoSplice."step".action1[3080] AND NOT false AND NOT false);
   "Unit1.Em2.ControlNodes".cmTapeTopUpDown.commands.commandWorkPos := NOT (NOT "Unit1.Em2.ControlNodes".semiAutoSplice."step".action1[2501] AND NOT "Unit1.Em2.ControlNodes".semiAutoSplice."step".action1[3076] AND NOT false AND NOT false AND NOT false);
END_REGION

REGION Network 79: Call instcmTapeTopUpDown (LBC_TwoWayActuator)
   RUNG wire#powerrail
      #instcmTapeTopUpDown(enable := TRUE, parentReferenceDesignator := "Unit1.Em2.Config".em.referenceDesignator.combined, feedbackHomePos := "BA030AZSBK02.03", feedbackWorkPos := "BA030AZSBK02.13", enableManualCmds := #statEnableManualCmds, interlockWorkPos := "Unit1.Em2.ControlNodes".cm.Interlock.tapeTopUpDown.work, interlockHomePos := "Unit1.Em2.ControlNodes".cm.Interlock.tapeTopUpDown.home, configuration := "Unit1.Em2.Config".cmTapeTopUpDown, moduleInterface := "Unit1.Em2.HmiInterface".cmTapeTopUpDown, controlNode := "Unit1.Em2.ControlNodes".cmTapeTopUpDown, goToHomePos => "BA030AZSPM02.07", goToWorkPos => "BA030AZSPM02.06")
   END_RUNG
   // the same network as SCL:
   #instcmTapeTopUpDown(enable := TRUE,   // "LBC_TwoWayActuatorCn"
                        parentReferenceDesignator := "Unit1.Em2.Config".em.referenceDesignator.combined,
                        feedbackHomePos := "BA030AZSBK02.03",
                        feedbackWorkPos := "BA030AZSBK02.13",
                        enableManualCmds := #statEnableManualCmds,
                        interlockWorkPos := "Unit1.Em2.ControlNodes".cm.Interlock.tapeTopUpDown.work,
                        interlockHomePos := "Unit1.Em2.ControlNodes".cm.Interlock.tapeTopUpDown.home,
                        configuration := "Unit1.Em2.Config".cmTapeTopUpDown,
                        moduleInterface := "Unit1.Em2.HmiInterface".cmTapeTopUpDown,
                        controlNode := "Unit1.Em2.ControlNodes".cmTapeTopUpDown,
                        goToHomePos => "BA030AZSPM02.07",
                        goToWorkPos => "BA030AZSPM02.06");
END_REGION

REGION Network 81: cmTapeBtmUpDown Interlock
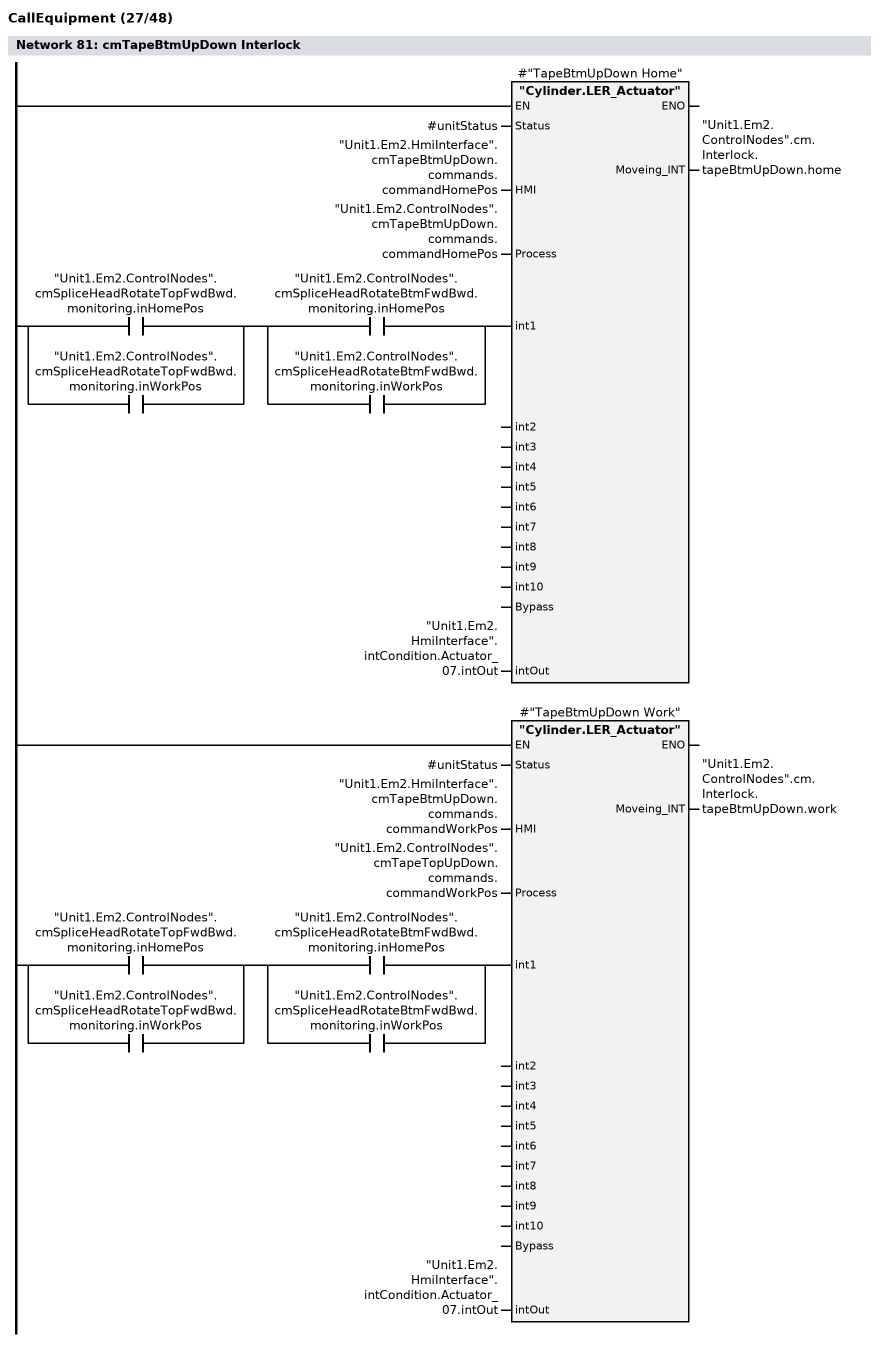
   RUNG wire#powerrail
      #"TapeBtmUpDown Home"(int1 := wire#w2, Status := #unitStatus, HMI := "Unit1.Em2.HmiInterface".cmTapeBtmUpDown.commands.commandHomePos, Process := "Unit1.Em2.ControlNodes".cmTapeBtmUpDown.commands.commandHomePos, int2 :=, int3 :=, int4 :=, int5 :=, int6 :=, int7 :=, int8 :=, int9 :=, int10 :=, Bypass :=, intOut := "Unit1.Em2.HmiInterface".intCondition.Actuator_07.intOut, Moveing_INT => "Unit1.Em2.ControlNodes".cm.Interlock.tapeBtmUpDown.home)
   END_RUNG
   RUNG wire#powerrail
      Contact( "Unit1.Em2.ControlNodes".cmSpliceHeadRotateTopFwdBwd.monitoring.inHomePos )
      wire#w1
      Contact( "Unit1.Em2.ControlNodes".cmSpliceHeadRotateBtmFwdBwd.monitoring.inHomePos )
   END_RUNG wire#w2
   RUNG wire#powerrail
      Contact( "Unit1.Em2.ControlNodes".cmSpliceHeadRotateTopFwdBwd.monitoring.inWorkPos )
   END_RUNG wire#w1
   RUNG wire#w1
      Contact( "Unit1.Em2.ControlNodes".cmSpliceHeadRotateBtmFwdBwd.monitoring.inWorkPos )
   END_RUNG wire#w2
   RUNG wire#powerrail
      #"TapeBtmUpDown Work"(int1 := wire#w4, Status := #unitStatus, HMI := "Unit1.Em2.HmiInterface".cmTapeBtmUpDown.commands.commandWorkPos, Process := "Unit1.Em2.ControlNodes".cmTapeTopUpDown.commands.commandWorkPos, int2 :=, int3 :=, int4 :=, int5 :=, int6 :=, int7 :=, int8 :=, int9 :=, int10 :=, Bypass :=, intOut := "Unit1.Em2.HmiInterface".intCondition.Actuator_07.intOut, Moveing_INT => "Unit1.Em2.ControlNodes".cm.Interlock.tapeBtmUpDown.work)
   END_RUNG
   RUNG wire#powerrail
      Contact( "Unit1.Em2.ControlNodes".cmSpliceHeadRotateTopFwdBwd.monitoring.inHomePos )
      wire#w3
      Contact( "Unit1.Em2.ControlNodes".cmSpliceHeadRotateBtmFwdBwd.monitoring.inHomePos )
   END_RUNG wire#w4
   RUNG wire#powerrail
      Contact( "Unit1.Em2.ControlNodes".cmSpliceHeadRotateTopFwdBwd.monitoring.inWorkPos )
   END_RUNG wire#w3
   RUNG wire#w3
      Contact( "Unit1.Em2.ControlNodes".cmSpliceHeadRotateBtmFwdBwd.monitoring.inWorkPos )
   END_RUNG wire#w4
   // the same network as SCL:
   #"TapeBtmUpDown Home"(Status := #unitStatus,   // "Cylinder.LER_Actuator"
                         HMI := "Unit1.Em2.HmiInterface".cmTapeBtmUpDown.commands.commandHomePos,
                         Process := "Unit1.Em2.ControlNodes".cmTapeBtmUpDown.commands.commandHomePos,
                         int1 := ("Unit1.Em2.ControlNodes".cmSpliceHeadRotateTopFwdBwd.monitoring.inHomePos OR "Unit1.Em2.ControlNodes".cmSpliceHeadRotateTopFwdBwd.monitoring.inWorkPos) AND ("Unit1.Em2.ControlNodes".cmSpliceHeadRotateBtmFwdBwd.monitoring.inHomePos OR "Unit1.Em2.ControlNodes".cmSpliceHeadRotateBtmFwdBwd.monitoring.inWorkPos),
                         intOut := "Unit1.Em2.HmiInterface".intCondition.Actuator_07.intOut,
                         Moveing_INT => "Unit1.Em2.ControlNodes".cm.Interlock.tapeBtmUpDown.home);
   #"TapeBtmUpDown Work"(Status := #unitStatus,   // "Cylinder.LER_Actuator"
                         HMI := "Unit1.Em2.HmiInterface".cmTapeBtmUpDown.commands.commandWorkPos,
                         Process := "Unit1.Em2.ControlNodes".cmTapeTopUpDown.commands.commandWorkPos,
                         int1 := ("Unit1.Em2.ControlNodes".cmSpliceHeadRotateTopFwdBwd.monitoring.inHomePos OR "Unit1.Em2.ControlNodes".cmSpliceHeadRotateTopFwdBwd.monitoring.inWorkPos) AND ("Unit1.Em2.ControlNodes".cmSpliceHeadRotateBtmFwdBwd.monitoring.inHomePos OR "Unit1.Em2.ControlNodes".cmSpliceHeadRotateBtmFwdBwd.monitoring.inWorkPos),
                         intOut := "Unit1.Em2.HmiInterface".intCondition.Actuator_07.intOut,
                         Moveing_INT => "Unit1.Em2.ControlNodes".cm.Interlock.tapeBtmUpDown.work);
END_REGION

REGION Network 82: cmTapeBtmUpDown Commands
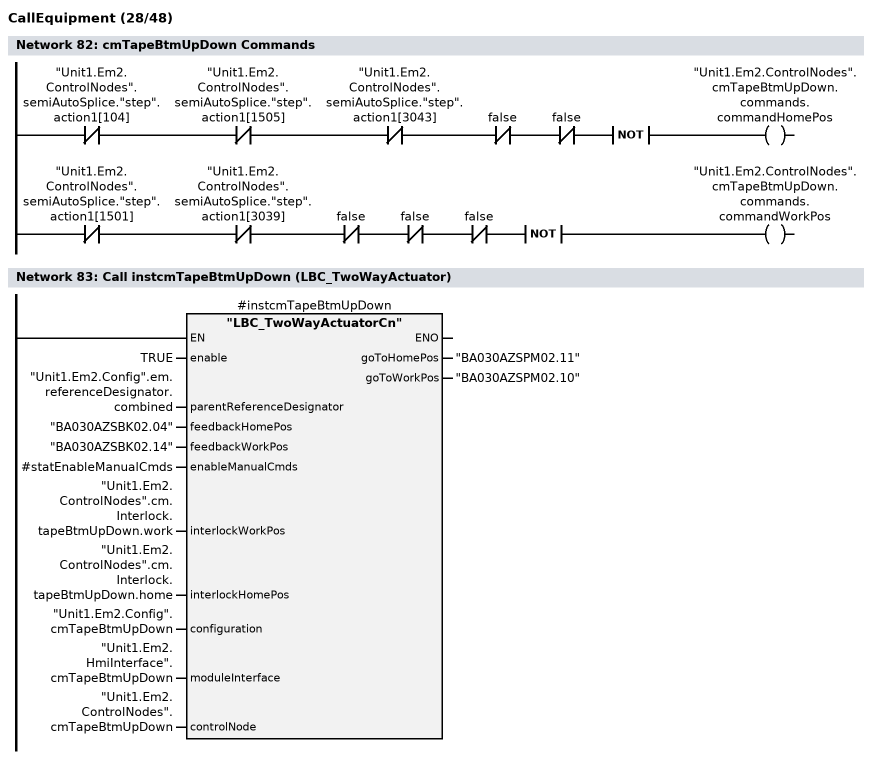
   RUNG wire#powerrail
      I_Contact( "Unit1.Em2.ControlNodes".semiAutoSplice."step".action1[104] )
      I_Contact( "Unit1.Em2.ControlNodes".semiAutoSplice."step".action1[1505] )
      I_Contact( "Unit1.Em2.ControlNodes".semiAutoSplice."step".action1[3043] )
      I_Contact( false )
      I_Contact( false )
      Not()
      Coil( "Unit1.Em2.ControlNodes".cmTapeBtmUpDown.commands.commandHomePos )
   END_RUNG
   RUNG wire#powerrail
      I_Contact( "Unit1.Em2.ControlNodes".semiAutoSplice."step".action1[1501] )
      I_Contact( "Unit1.Em2.ControlNodes".semiAutoSplice."step".action1[3039] )
      I_Contact( false )
      I_Contact( false )
      I_Contact( false )
      Not()
      Coil( "Unit1.Em2.ControlNodes".cmTapeBtmUpDown.commands.commandWorkPos )
   END_RUNG
   // the same network as SCL:
   "Unit1.Em2.ControlNodes".cmTapeBtmUpDown.commands.commandHomePos := NOT (NOT "Unit1.Em2.ControlNodes".semiAutoSplice."step".action1[104] AND NOT "Unit1.Em2.ControlNodes".semiAutoSplice."step".action1[1505] AND NOT "Unit1.Em2.ControlNodes".semiAutoSplice."step".action1[3043] AND NOT false AND NOT false);
   "Unit1.Em2.ControlNodes".cmTapeBtmUpDown.commands.commandWorkPos := NOT (NOT "Unit1.Em2.ControlNodes".semiAutoSplice."step".action1[1501] AND NOT "Unit1.Em2.ControlNodes".semiAutoSplice."step".action1[3039] AND NOT false AND NOT false AND NOT false);
END_REGION

REGION Network 83: Call instcmTapeBtmUpDown (LBC_TwoWayActuator)
   RUNG wire#powerrail
      #instcmTapeBtmUpDown(enable := TRUE, parentReferenceDesignator := "Unit1.Em2.Config".em.referenceDesignator.combined, feedbackHomePos := "BA030AZSBK02.04", feedbackWorkPos := "BA030AZSBK02.14", enableManualCmds := #statEnableManualCmds, interlockWorkPos := "Unit1.Em2.ControlNodes".cm.Interlock.tapeBtmUpDown.work, interlockHomePos := "Unit1.Em2.ControlNodes".cm.Interlock.tapeBtmUpDown.home, configuration := "Unit1.Em2.Config".cmTapeBtmUpDown, moduleInterface := "Unit1.Em2.HmiInterface".cmTapeBtmUpDown, controlNode := "Unit1.Em2.ControlNodes".cmTapeBtmUpDown, goToHomePos => "BA030AZSPM02.11", goToWorkPos => "BA030AZSPM02.10")
   END_RUNG
   // the same network as SCL:
   #instcmTapeBtmUpDown(enable := TRUE,   // "LBC_TwoWayActuatorCn"
                        parentReferenceDesignator := "Unit1.Em2.Config".em.referenceDesignator.combined,
                        feedbackHomePos := "BA030AZSBK02.04",
                        feedbackWorkPos := "BA030AZSBK02.14",
                        enableManualCmds := #statEnableManualCmds,
                        interlockWorkPos := "Unit1.Em2.ControlNodes".cm.Interlock.tapeBtmUpDown.work,
                        interlockHomePos := "Unit1.Em2.ControlNodes".cm.Interlock.tapeBtmUpDown.home,
                        configuration := "Unit1.Em2.Config".cmTapeBtmUpDown,
                        moduleInterface := "Unit1.Em2.HmiInterface".cmTapeBtmUpDown,
                        controlNode := "Unit1.Em2.ControlNodes".cmTapeBtmUpDown,
                        goToHomePos => "BA030AZSPM02.11",
                        goToWorkPos => "BA030AZSPM02.10");
END_REGION

REGION Network 85: cmSpliceHeadRotateTopFwdBwd Interlock
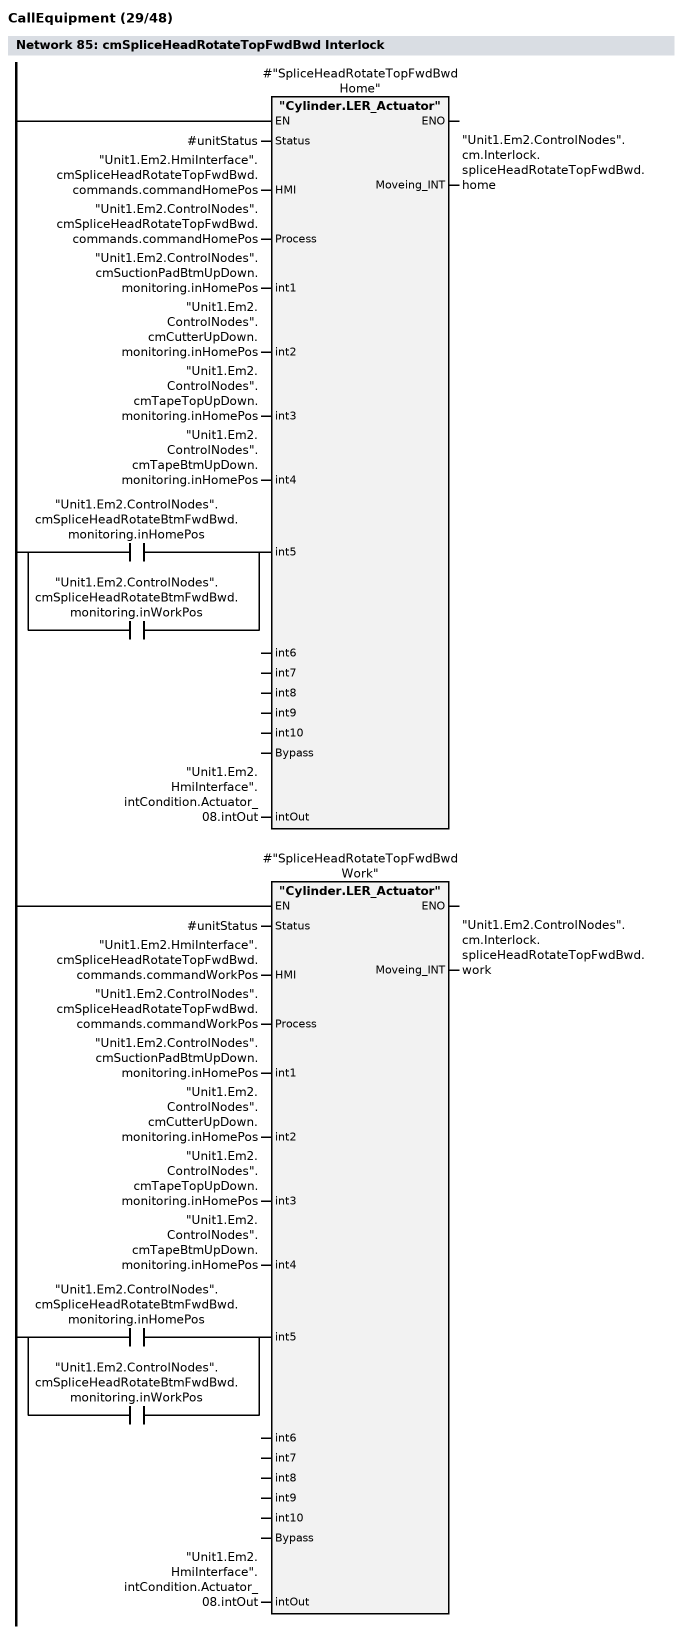
   RUNG wire#powerrail
      #"SpliceHeadRotateTopFwdBwd Home"(int5 := wire#w1, Status := #unitStatus, HMI := "Unit1.Em2.HmiInterface".cmSpliceHeadRotateTopFwdBwd.commands.commandHomePos, Process := "Unit1.Em2.ControlNodes".cmSpliceHeadRotateTopFwdBwd.commands.commandHomePos, int1 := "Unit1.Em2.ControlNodes".cmSuctionPadBtmUpDown.monitoring.inHomePos, int2 := "Unit1.Em2.ControlNodes".cmCutterUpDown.monitoring.inHomePos, int3 := "Unit1.Em2.ControlNodes".cmTapeTopUpDown.monitoring.inHomePos, int4 := "Unit1.Em2.ControlNodes".cmTapeBtmUpDown.monitoring.inHomePos, int6 :=, int7 :=, int8 :=, int9 :=, int10 :=, Bypass :=, intOut := "Unit1.Em2.HmiInterface".intCondition.Actuator_08.intOut, Moveing_INT => "Unit1.Em2.ControlNodes".cm.Interlock.spliceHeadRotateTopFwdBwd.home)
   END_RUNG
   RUNG wire#powerrail
      Contact( "Unit1.Em2.ControlNodes".cmSpliceHeadRotateBtmFwdBwd.monitoring.inHomePos )
   END_RUNG wire#w1
   RUNG wire#powerrail
      Contact( "Unit1.Em2.ControlNodes".cmSpliceHeadRotateBtmFwdBwd.monitoring.inWorkPos )
   END_RUNG wire#w1
   RUNG wire#powerrail
      #"SpliceHeadRotateTopFwdBwd Work"(int5 := wire#w2, Status := #unitStatus, HMI := "Unit1.Em2.HmiInterface".cmSpliceHeadRotateTopFwdBwd.commands.commandWorkPos, Process := "Unit1.Em2.ControlNodes".cmSpliceHeadRotateTopFwdBwd.commands.commandWorkPos, int1 := "Unit1.Em2.ControlNodes".cmSuctionPadBtmUpDown.monitoring.inHomePos, int2 := "Unit1.Em2.ControlNodes".cmCutterUpDown.monitoring.inHomePos, int3 := "Unit1.Em2.ControlNodes".cmTapeTopUpDown.monitoring.inHomePos, int4 := "Unit1.Em2.ControlNodes".cmTapeBtmUpDown.monitoring.inHomePos, int6 :=, int7 :=, int8 :=, int9 :=, int10 :=, Bypass :=, intOut := "Unit1.Em2.HmiInterface".intCondition.Actuator_08.intOut, Moveing_INT => "Unit1.Em2.ControlNodes".cm.Interlock.spliceHeadRotateTopFwdBwd.work)
   END_RUNG
   RUNG wire#powerrail
      Contact( "Unit1.Em2.ControlNodes".cmSpliceHeadRotateBtmFwdBwd.monitoring.inHomePos )
   END_RUNG wire#w2
   RUNG wire#powerrail
      Contact( "Unit1.Em2.ControlNodes".cmSpliceHeadRotateBtmFwdBwd.monitoring.inWorkPos )
   END_RUNG wire#w2
   // the same network as SCL:
   #"SpliceHeadRotateTopFwdBwd Home"(Status := #unitStatus,   // "Cylinder.LER_Actuator"
                           HMI := "Unit1.Em2.HmiInterface".cmSpliceHeadRotateTopFwdBwd.commands.commandHomePos,
                           Process := "Unit1.Em2.ControlNodes".cmSpliceHeadRotateTopFwdBwd.commands.commandHomePos,
                           int1 := "Unit1.Em2.ControlNodes".cmSuctionPadBtmUpDown.monitoring.inHomePos,
                           int2 := "Unit1.Em2.ControlNodes".cmCutterUpDown.monitoring.inHomePos,
                           int3 := "Unit1.Em2.ControlNodes".cmTapeTopUpDown.monitoring.inHomePos,
                           int4 := "Unit1.Em2.ControlNodes".cmTapeBtmUpDown.monitoring.inHomePos,
                           int5 := "Unit1.Em2.ControlNodes".cmSpliceHeadRotateBtmFwdBwd.monitoring.inHomePos OR "Unit1.Em2.ControlNodes".cmSpliceHeadRotateBtmFwdBwd.monitoring.inWorkPos,
                           intOut := "Unit1.Em2.HmiInterface".intCondition.Actuator_08.intOut,
                           Moveing_INT => "Unit1.Em2.ControlNodes".cm.Interlock.spliceHeadRotateTopFwdBwd.home);
   #"SpliceHeadRotateTopFwdBwd Work"(Status := #unitStatus,   // "Cylinder.LER_Actuator"
                           HMI := "Unit1.Em2.HmiInterface".cmSpliceHeadRotateTopFwdBwd.commands.commandWorkPos,
                           Process := "Unit1.Em2.ControlNodes".cmSpliceHeadRotateTopFwdBwd.commands.commandWorkPos,
                           int1 := "Unit1.Em2.ControlNodes".cmSuctionPadBtmUpDown.monitoring.inHomePos,
                           int2 := "Unit1.Em2.ControlNodes".cmCutterUpDown.monitoring.inHomePos,
                           int3 := "Unit1.Em2.ControlNodes".cmTapeTopUpDown.monitoring.inHomePos,
                           int4 := "Unit1.Em2.ControlNodes".cmTapeBtmUpDown.monitoring.inHomePos,
                           int5 := "Unit1.Em2.ControlNodes".cmSpliceHeadRotateBtmFwdBwd.monitoring.inHomePos OR "Unit1.Em2.ControlNodes".cmSpliceHeadRotateBtmFwdBwd.monitoring.inWorkPos,
                           intOut := "Unit1.Em2.HmiInterface".intCondition.Actuator_08.intOut,
                           Moveing_INT => "Unit1.Em2.ControlNodes".cm.Interlock.spliceHeadRotateTopFwdBwd.work);
END_REGION

REGION Network 86: cmSpliceHeadRotateTopFwdBwd Commmands
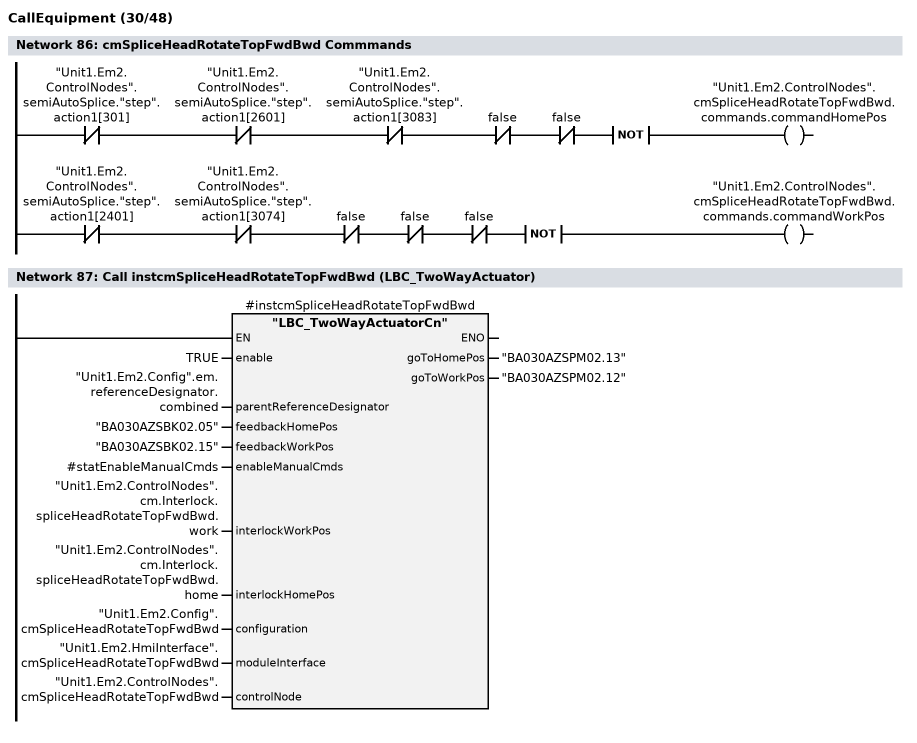
   RUNG wire#powerrail
      I_Contact( "Unit1.Em2.ControlNodes".semiAutoSplice."step".action1[301] )
      I_Contact( "Unit1.Em2.ControlNodes".semiAutoSplice."step".action1[2601] )
      I_Contact( "Unit1.Em2.ControlNodes".semiAutoSplice."step".action1[3083] )
      I_Contact( false )
      I_Contact( false )
      Not()
      Coil( "Unit1.Em2.ControlNodes".cmSpliceHeadRotateTopFwdBwd.commands.commandHomePos )
   END_RUNG
   RUNG wire#powerrail
      I_Contact( "Unit1.Em2.ControlNodes".semiAutoSplice."step".action1[2401] )
      I_Contact( "Unit1.Em2.ControlNodes".semiAutoSplice."step".action1[3074] )
      I_Contact( false )
      I_Contact( false )
      I_Contact( false )
      Not()
      Coil( "Unit1.Em2.ControlNodes".cmSpliceHeadRotateTopFwdBwd.commands.commandWorkPos )
   END_RUNG
   // the same network as SCL:
   "Unit1.Em2.ControlNodes".cmSpliceHeadRotateTopFwdBwd.commands.commandHomePos := NOT (NOT "Unit1.Em2.ControlNodes".semiAutoSplice."step".action1[301] AND NOT "Unit1.Em2.ControlNodes".semiAutoSplice."step".action1[2601] AND NOT "Unit1.Em2.ControlNodes".semiAutoSplice."step".action1[3083] AND NOT false AND NOT false);
   "Unit1.Em2.ControlNodes".cmSpliceHeadRotateTopFwdBwd.commands.commandWorkPos := NOT (NOT "Unit1.Em2.ControlNodes".semiAutoSplice."step".action1[2401] AND NOT "Unit1.Em2.ControlNodes".semiAutoSplice."step".action1[3074] AND NOT false AND NOT false AND NOT false);
END_REGION

REGION Network 87: Call instcmSpliceHeadRotateTopFwdBwd (LBC_TwoWayActuator)
   RUNG wire#powerrail
      #instcmSpliceHeadRotateTopFwdBwd(enable := TRUE, parentReferenceDesignator := "Unit1.Em2.Config".em.referenceDesignator.combined, feedbackHomePos := "BA030AZSBK02.05", feedbackWorkPos := "BA030AZSBK02.15", enableManualCmds := #statEnableManualCmds, interlockWorkPos := "Unit1.Em2.ControlNodes".cm.Interlock.spliceHeadRotateTopFwdBwd.work, interlockHomePos := "Unit1.Em2.ControlNodes".cm.Interlock.spliceHeadRotateTopFwdBwd.home, configuration := "Unit1.Em2.Config".cmSpliceHeadRotateTopFwdBwd, moduleInterface := "Unit1.Em2.HmiInterface".cmSpliceHeadRotateTopFwdBwd, controlNode := "Unit1.Em2.ControlNodes".cmSpliceHeadRotateTopFwdBwd, goToHomePos => "BA030AZSPM02.13", goToWorkPos => "BA030AZSPM02.12")
   END_RUNG
   // the same network as SCL:
   #instcmSpliceHeadRotateTopFwdBwd(enable := TRUE,   // "LBC_TwoWayActuatorCn"
                           parentReferenceDesignator := "Unit1.Em2.Config".em.referenceDesignator.combined,
                           feedbackHomePos := "BA030AZSBK02.05",
                           feedbackWorkPos := "BA030AZSBK02.15",
                           enableManualCmds := #statEnableManualCmds,
                           interlockWorkPos := "Unit1.Em2.ControlNodes".cm.Interlock.spliceHeadRotateTopFwdBwd.work,
                           interlockHomePos := "Unit1.Em2.ControlNodes".cm.Interlock.spliceHeadRotateTopFwdBwd.home,
                           configuration := "Unit1.Em2.Config".cmSpliceHeadRotateTopFwdBwd,
                           moduleInterface := "Unit1.Em2.HmiInterface".cmSpliceHeadRotateTopFwdBwd,
                           controlNode := "Unit1.Em2.ControlNodes".cmSpliceHeadRotateTopFwdBwd,
                           goToHomePos => "BA030AZSPM02.13",
                           goToWorkPos => "BA030AZSPM02.12");
END_REGION

REGION Network 89: cmSpliceHeadRotateBtmFwdBwd Interlock
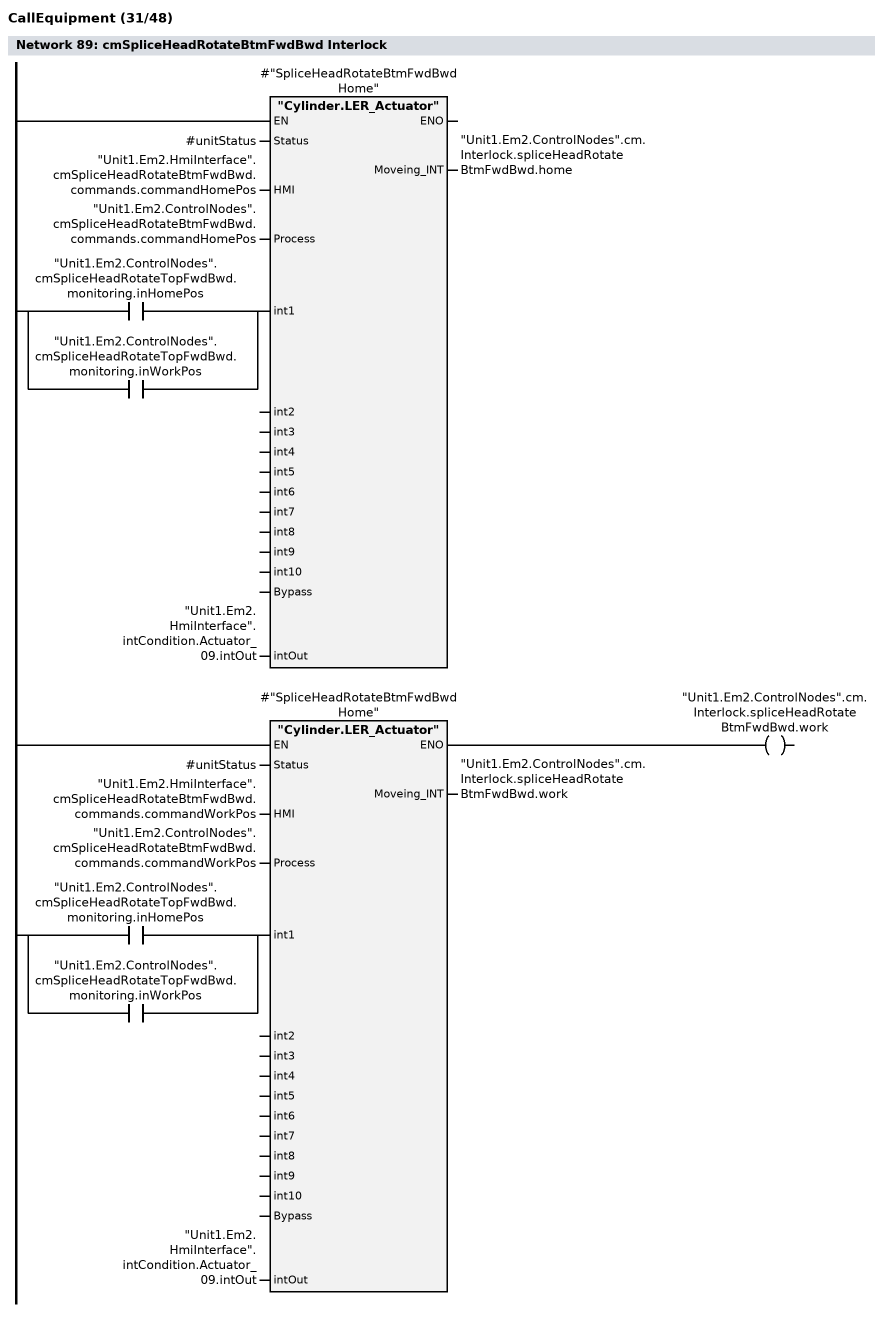
   RUNG wire#powerrail
      #"SpliceHeadRotateBtmFwdBwd Home"(int1 := wire#w1, Status := #unitStatus, HMI := "Unit1.Em2.HmiInterface".cmSpliceHeadRotateBtmFwdBwd.commands.commandHomePos, Process := "Unit1.Em2.ControlNodes".cmSpliceHeadRotateBtmFwdBwd.commands.commandHomePos, int2 :=, int3 :=, int4 :=, int5 :=, int6 :=, int7 :=, int8 :=, int9 :=, int10 :=, Bypass :=, intOut := "Unit1.Em2.HmiInterface".intCondition.Actuator_09.intOut, Moveing_INT => "Unit1.Em2.ControlNodes".cm.Interlock.spliceHeadRotateBtmFwdBwd.home)
   END_RUNG
   RUNG wire#powerrail
      Contact( "Unit1.Em2.ControlNodes".cmSpliceHeadRotateTopFwdBwd.monitoring.inHomePos )
   END_RUNG wire#w1
   RUNG wire#powerrail
      Contact( "Unit1.Em2.ControlNodes".cmSpliceHeadRotateTopFwdBwd.monitoring.inWorkPos )
   END_RUNG wire#w1
   RUNG wire#powerrail
      #"SpliceHeadRotateBtmFwdBwd Home"(int1 := wire#w2, Status := #unitStatus, HMI := "Unit1.Em2.HmiInterface".cmSpliceHeadRotateBtmFwdBwd.commands.commandWorkPos, Process := "Unit1.Em2.ControlNodes".cmSpliceHeadRotateBtmFwdBwd.commands.commandWorkPos, int2 :=, int3 :=, int4 :=, int5 :=, int6 :=, int7 :=, int8 :=, int9 :=, int10 :=, Bypass :=, intOut := "Unit1.Em2.HmiInterface".intCondition.Actuator_09.intOut, Moveing_INT => "Unit1.Em2.ControlNodes".cm.Interlock.spliceHeadRotateBtmFwdBwd.work)
      Coil( "Unit1.Em2.ControlNodes".cm.Interlock.spliceHeadRotateBtmFwdBwd.work )
   END_RUNG
   RUNG wire#powerrail
      Contact( "Unit1.Em2.ControlNodes".cmSpliceHeadRotateTopFwdBwd.monitoring.inHomePos )
   END_RUNG wire#w2
   RUNG wire#powerrail
      Contact( "Unit1.Em2.ControlNodes".cmSpliceHeadRotateTopFwdBwd.monitoring.inWorkPos )
   END_RUNG wire#w2
   // the same network as SCL:
   #"SpliceHeadRotateBtmFwdBwd Home"(Status := #unitStatus,   // "Cylinder.LER_Actuator"
                           HMI := "Unit1.Em2.HmiInterface".cmSpliceHeadRotateBtmFwdBwd.commands.commandHomePos,
                           Process := "Unit1.Em2.ControlNodes".cmSpliceHeadRotateBtmFwdBwd.commands.commandHomePos,
                           int1 := "Unit1.Em2.ControlNodes".cmSpliceHeadRotateTopFwdBwd.monitoring.inHomePos OR "Unit1.Em2.ControlNodes".cmSpliceHeadRotateTopFwdBwd.monitoring.inWorkPos,
                           intOut := "Unit1.Em2.HmiInterface".intCondition.Actuator_09.intOut,
                           Moveing_INT => "Unit1.Em2.ControlNodes".cm.Interlock.spliceHeadRotateBtmFwdBwd.home);
   #"SpliceHeadRotateBtmFwdBwd Home"(Status := #unitStatus,   // "Cylinder.LER_Actuator"
                           HMI := "Unit1.Em2.HmiInterface".cmSpliceHeadRotateBtmFwdBwd.commands.commandWorkPos,
                           Process := "Unit1.Em2.ControlNodes".cmSpliceHeadRotateBtmFwdBwd.commands.commandWorkPos,
                           int1 := "Unit1.Em2.ControlNodes".cmSpliceHeadRotateTopFwdBwd.monitoring.inHomePos OR "Unit1.Em2.ControlNodes".cmSpliceHeadRotateTopFwdBwd.monitoring.inWorkPos,
                           intOut := "Unit1.Em2.HmiInterface".intCondition.Actuator_09.intOut,
                           Moveing_INT => "Unit1.Em2.ControlNodes".cm.Interlock.spliceHeadRotateBtmFwdBwd.work,
                           ENO => #_w1);
   "Unit1.Em2.ControlNodes".cm.Interlock.spliceHeadRotateBtmFwdBwd.work := #_w1;
END_REGION

REGION Network 90: cmSpliceHeadRotateBtmFwdBwd Commands
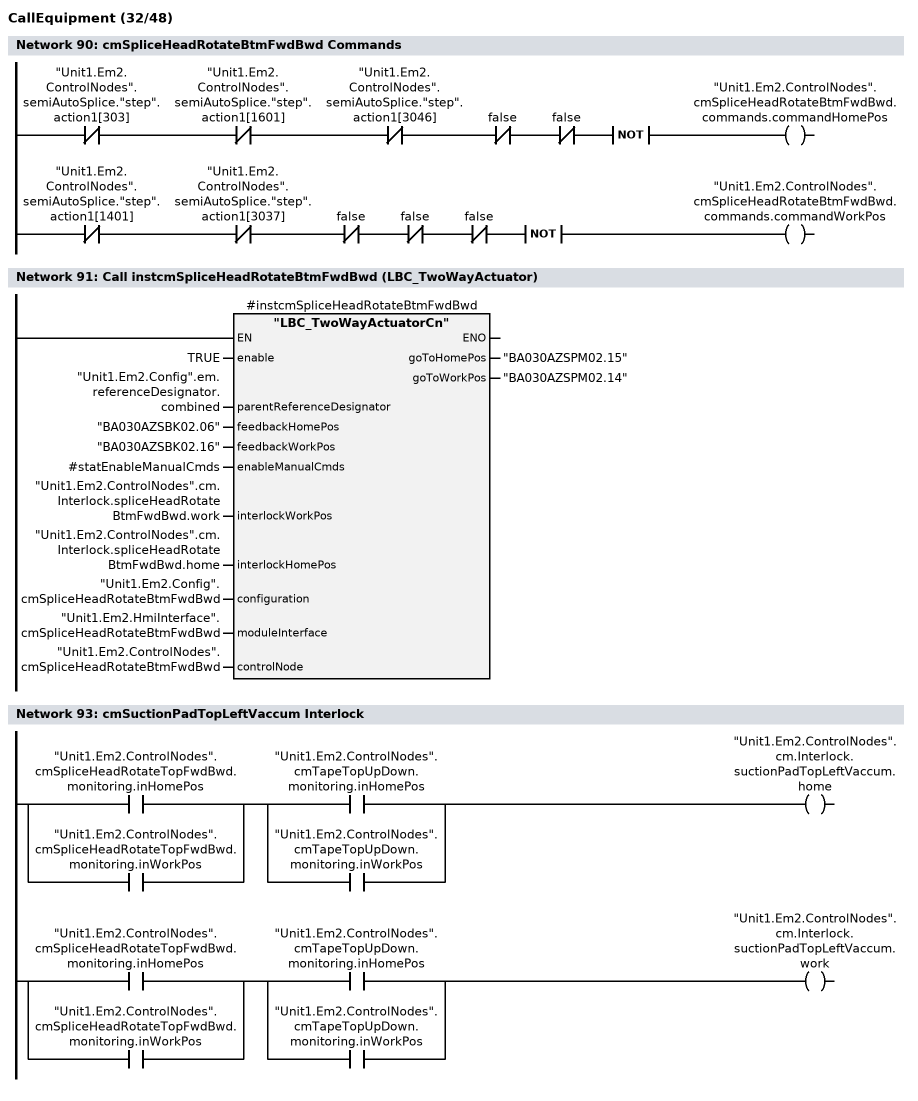
   RUNG wire#powerrail
      I_Contact( "Unit1.Em2.ControlNodes".semiAutoSplice."step".action1[303] )
      I_Contact( "Unit1.Em2.ControlNodes".semiAutoSplice."step".action1[1601] )
      I_Contact( "Unit1.Em2.ControlNodes".semiAutoSplice."step".action1[3046] )
      I_Contact( false )
      I_Contact( false )
      Not()
      Coil( "Unit1.Em2.ControlNodes".cmSpliceHeadRotateBtmFwdBwd.commands.commandHomePos )
   END_RUNG
   RUNG wire#powerrail
      I_Contact( "Unit1.Em2.ControlNodes".semiAutoSplice."step".action1[1401] )
      I_Contact( "Unit1.Em2.ControlNodes".semiAutoSplice."step".action1[3037] )
      I_Contact( false )
      I_Contact( false )
      I_Contact( false )
      Not()
      Coil( "Unit1.Em2.ControlNodes".cmSpliceHeadRotateBtmFwdBwd.commands.commandWorkPos )
   END_RUNG
   // the same network as SCL:
   "Unit1.Em2.ControlNodes".cmSpliceHeadRotateBtmFwdBwd.commands.commandHomePos := NOT (NOT "Unit1.Em2.ControlNodes".semiAutoSplice."step".action1[303] AND NOT "Unit1.Em2.ControlNodes".semiAutoSplice."step".action1[1601] AND NOT "Unit1.Em2.ControlNodes".semiAutoSplice."step".action1[3046] AND NOT false AND NOT false);
   "Unit1.Em2.ControlNodes".cmSpliceHeadRotateBtmFwdBwd.commands.commandWorkPos := NOT (NOT "Unit1.Em2.ControlNodes".semiAutoSplice."step".action1[1401] AND NOT "Unit1.Em2.ControlNodes".semiAutoSplice."step".action1[3037] AND NOT false AND NOT false AND NOT false);
END_REGION

REGION Network 91: Call instcmSpliceHeadRotateBtmFwdBwd (LBC_TwoWayActuator)
   RUNG wire#powerrail
      #instcmSpliceHeadRotateBtmFwdBwd(enable := TRUE, parentReferenceDesignator := "Unit1.Em2.Config".em.referenceDesignator.combined, feedbackHomePos := "BA030AZSBK02.06", feedbackWorkPos := "BA030AZSBK02.16", enableManualCmds := #statEnableManualCmds, interlockWorkPos := "Unit1.Em2.ControlNodes".cm.Interlock.spliceHeadRotateBtmFwdBwd.work, interlockHomePos := "Unit1.Em2.ControlNodes".cm.Interlock.spliceHeadRotateBtmFwdBwd.home, configuration := "Unit1.Em2.Config".cmSpliceHeadRotateBtmFwdBwd, moduleInterface := "Unit1.Em2.HmiInterface".cmSpliceHeadRotateBtmFwdBwd, controlNode := "Unit1.Em2.ControlNodes".cmSpliceHeadRotateBtmFwdBwd, goToHomePos => "BA030AZSPM02.15", goToWorkPos => "BA030AZSPM02.14")
   END_RUNG
   // the same network as SCL:
   #instcmSpliceHeadRotateBtmFwdBwd(enable := TRUE,   // "LBC_TwoWayActuatorCn"
                           parentReferenceDesignator := "Unit1.Em2.Config".em.referenceDesignator.combined,
                           feedbackHomePos := "BA030AZSBK02.06",
                           feedbackWorkPos := "BA030AZSBK02.16",
                           enableManualCmds := #statEnableManualCmds,
                           interlockWorkPos := "Unit1.Em2.ControlNodes".cm.Interlock.spliceHeadRotateBtmFwdBwd.work,
                           interlockHomePos := "Unit1.Em2.ControlNodes".cm.Interlock.spliceHeadRotateBtmFwdBwd.home,
                           configuration := "Unit1.Em2.Config".cmSpliceHeadRotateBtmFwdBwd,
                           moduleInterface := "Unit1.Em2.HmiInterface".cmSpliceHeadRotateBtmFwdBwd,
                           controlNode := "Unit1.Em2.ControlNodes".cmSpliceHeadRotateBtmFwdBwd,
                           goToHomePos => "BA030AZSPM02.15",
                           goToWorkPos => "BA030AZSPM02.14");
END_REGION

REGION Network 93: cmSuctionPadTopLeftVaccum Interlock
   RUNG wire#powerrail
      Contact( "Unit1.Em2.ControlNodes".cmSpliceHeadRotateTopFwdBwd.monitoring.inHomePos )
      wire#w1
      Contact( "Unit1.Em2.ControlNodes".cmTapeTopUpDown.monitoring.inHomePos )
      wire#w2
      Coil( "Unit1.Em2.ControlNodes".cm.Interlock.suctionPadTopLeftVaccum.home )
   END_RUNG
   RUNG wire#powerrail
      Contact( "Unit1.Em2.ControlNodes".cmSpliceHeadRotateTopFwdBwd.monitoring.inWorkPos )
   END_RUNG wire#w1
   RUNG wire#w1
      Contact( "Unit1.Em2.ControlNodes".cmTapeTopUpDown.monitoring.inWorkPos )
   END_RUNG wire#w2
   RUNG wire#powerrail
      Contact( "Unit1.Em2.ControlNodes".cmSpliceHeadRotateTopFwdBwd.monitoring.inHomePos )
      wire#w3
      Contact( "Unit1.Em2.ControlNodes".cmTapeTopUpDown.monitoring.inHomePos )
      wire#w4
      Coil( "Unit1.Em2.ControlNodes".cm.Interlock.suctionPadTopLeftVaccum.work )
   END_RUNG
   RUNG wire#powerrail
      Contact( "Unit1.Em2.ControlNodes".cmSpliceHeadRotateTopFwdBwd.monitoring.inWorkPos )
   END_RUNG wire#w3
   RUNG wire#w3
      Contact( "Unit1.Em2.ControlNodes".cmTapeTopUpDown.monitoring.inWorkPos )
   END_RUNG wire#w4
   // the same network as SCL:
   "Unit1.Em2.ControlNodes".cm.Interlock.suctionPadTopLeftVaccum.home := ("Unit1.Em2.ControlNodes".cmSpliceHeadRotateTopFwdBwd.monitoring.inHomePos OR "Unit1.Em2.ControlNodes".cmSpliceHeadRotateTopFwdBwd.monitoring.inWorkPos) AND ("Unit1.Em2.ControlNodes".cmTapeTopUpDown.monitoring.inHomePos OR "Unit1.Em2.ControlNodes".cmTapeTopUpDown.monitoring.inWorkPos);
   "Unit1.Em2.ControlNodes".cm.Interlock.suctionPadTopLeftVaccum.work := ("Unit1.Em2.ControlNodes".cmSpliceHeadRotateTopFwdBwd.monitoring.inHomePos OR "Unit1.Em2.ControlNodes".cmSpliceHeadRotateTopFwdBwd.monitoring.inWorkPos) AND ("Unit1.Em2.ControlNodes".cmTapeTopUpDown.monitoring.inHomePos OR "Unit1.Em2.ControlNodes".cmTapeTopUpDown.monitoring.inWorkPos);
END_REGION

REGION Network 94: cmSuctionPadTopLeftVaccum Commands
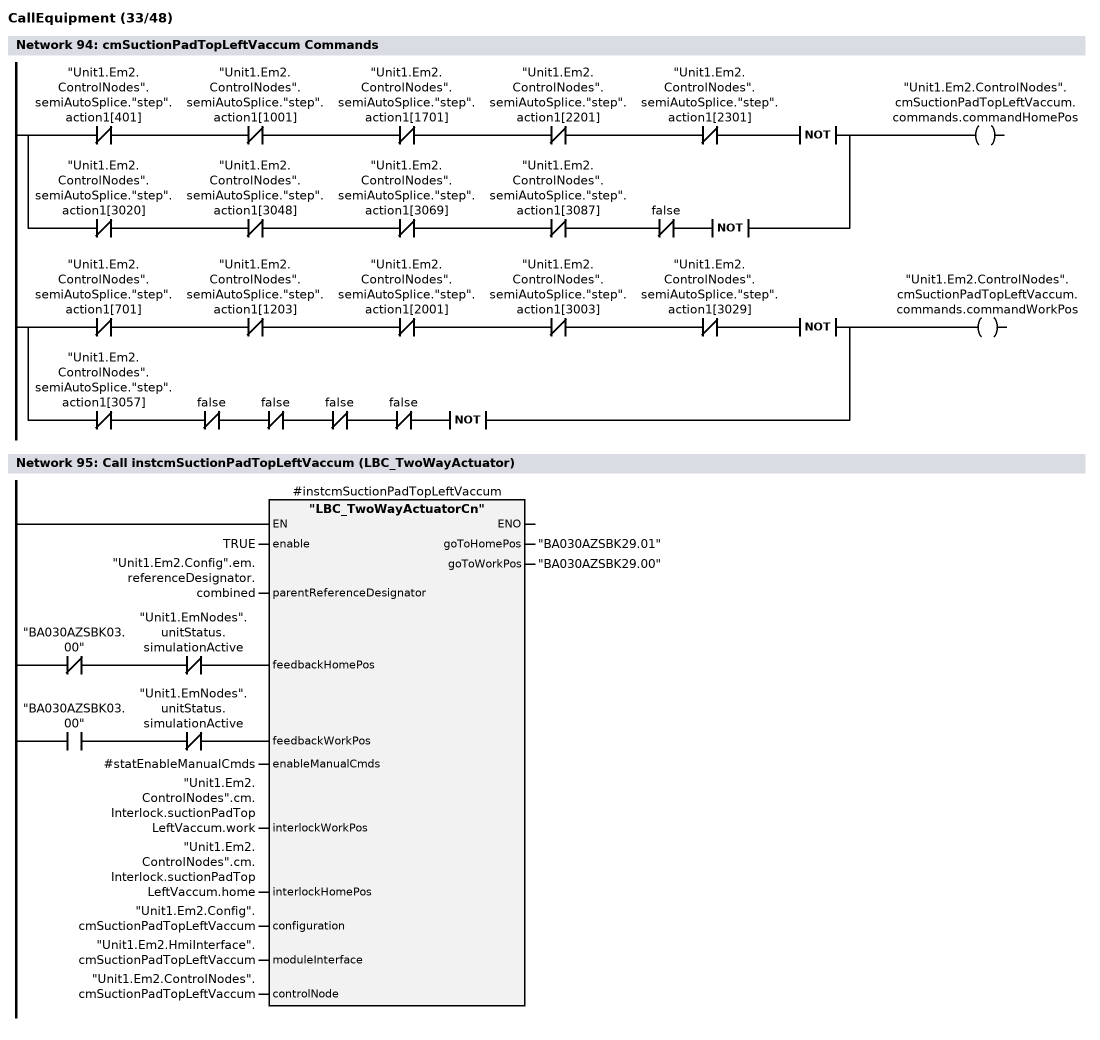
   RUNG wire#powerrail
      I_Contact( "Unit1.Em2.ControlNodes".semiAutoSplice."step".action1[401] )
      I_Contact( "Unit1.Em2.ControlNodes".semiAutoSplice."step".action1[1001] )
      I_Contact( "Unit1.Em2.ControlNodes".semiAutoSplice."step".action1[1701] )
      I_Contact( "Unit1.Em2.ControlNodes".semiAutoSplice."step".action1[2201] )
      I_Contact( "Unit1.Em2.ControlNodes".semiAutoSplice."step".action1[2301] )
      Not()
      wire#w1
      Coil( "Unit1.Em2.ControlNodes".cmSuctionPadTopLeftVaccum.commands.commandHomePos )
   END_RUNG
   RUNG wire#powerrail
      I_Contact( "Unit1.Em2.ControlNodes".semiAutoSplice."step".action1[3020] )
      I_Contact( "Unit1.Em2.ControlNodes".semiAutoSplice."step".action1[3048] )
      I_Contact( "Unit1.Em2.ControlNodes".semiAutoSplice."step".action1[3069] )
      I_Contact( "Unit1.Em2.ControlNodes".semiAutoSplice."step".action1[3087] )
      I_Contact( false )
      Not()
   END_RUNG wire#w1
   RUNG wire#powerrail
      I_Contact( "Unit1.Em2.ControlNodes".semiAutoSplice."step".action1[701] )
      I_Contact( "Unit1.Em2.ControlNodes".semiAutoSplice."step".action1[1203] )
      I_Contact( "Unit1.Em2.ControlNodes".semiAutoSplice."step".action1[2001] )
      I_Contact( "Unit1.Em2.ControlNodes".semiAutoSplice."step".action1[3003] )
      I_Contact( "Unit1.Em2.ControlNodes".semiAutoSplice."step".action1[3029] )
      Not()
      wire#w2
      Coil( "Unit1.Em2.ControlNodes".cmSuctionPadTopLeftVaccum.commands.commandWorkPos )
   END_RUNG
   RUNG wire#powerrail
      I_Contact( "Unit1.Em2.ControlNodes".semiAutoSplice."step".action1[3057] )
      I_Contact( false )
      I_Contact( false )
      I_Contact( false )
      I_Contact( false )
      Not()
   END_RUNG wire#w2
   // the same network as SCL:
   "Unit1.Em2.ControlNodes".cmSuctionPadTopLeftVaccum.commands.commandHomePos := NOT (NOT "Unit1.Em2.ControlNodes".semiAutoSplice."step".action1[401] AND NOT "Unit1.Em2.ControlNodes".semiAutoSplice."step".action1[1001] AND NOT "Unit1.Em2.ControlNodes".semiAutoSplice."step".action1[1701] AND NOT "Unit1.Em2.ControlNodes".semiAutoSplice."step".action1[2201] AND NOT "Unit1.Em2.ControlNodes".semiAutoSplice."step".action1[2301]) OR NOT (NOT "Unit1.Em2.ControlNodes".semiAutoSplice."step".action1[3020] AND NOT "Unit1.Em2.ControlNodes".semiAutoSplice."step".action1[3048] AND NOT "Unit1.Em2.ControlNodes".semiAutoSplice."step".action1[3069] AND NOT "Unit1.Em2.ControlNodes".semiAutoSplice."step".action1[3087] AND NOT false);
   "Unit1.Em2.ControlNodes".cmSuctionPadTopLeftVaccum.commands.commandWorkPos := NOT (NOT "Unit1.Em2.ControlNodes".semiAutoSplice."step".action1[701] AND NOT "Unit1.Em2.ControlNodes".semiAutoSplice."step".action1[1203] AND NOT "Unit1.Em2.ControlNodes".semiAutoSplice."step".action1[2001] AND NOT "Unit1.Em2.ControlNodes".semiAutoSplice."step".action1[3003] AND NOT "Unit1.Em2.ControlNodes".semiAutoSplice."step".action1[3029]) OR NOT (NOT "Unit1.Em2.ControlNodes".semiAutoSplice."step".action1[3057] AND NOT false AND NOT false AND NOT false AND NOT false);
END_REGION

REGION Network 95: Call instcmSuctionPadTopLeftVaccum (LBC_TwoWayActuator)
   RUNG wire#powerrail
      #instcmSuctionPadTopLeftVaccum(feedbackHomePos := wire#w1, feedbackWorkPos := wire#w2, enable := TRUE, parentReferenceDesignator := "Unit1.Em2.Config".em.referenceDesignator.combined, enableManualCmds := #statEnableManualCmds, interlockWorkPos := "Unit1.Em2.ControlNodes".cm.Interlock.suctionPadTopLeftVaccum.work, interlockHomePos := "Unit1.Em2.ControlNodes".cm.Interlock.suctionPadTopLeftVaccum.home, configuration := "Unit1.Em2.Config".cmSuctionPadTopLeftVaccum, moduleInterface := "Unit1.Em2.HmiInterface".cmSuctionPadTopLeftVaccum, controlNode := "Unit1.Em2.ControlNodes".cmSuctionPadTopLeftVaccum, goToHomePos => "BA030AZSBK29.01", goToWorkPos => "BA030AZSBK29.00")
   END_RUNG
   RUNG wire#powerrail
      I_Contact( "BA030AZSBK03.00" )
      I_Contact( "Unit1.EmNodes".unitStatus.simulationActive )
   END_RUNG wire#w1
   RUNG wire#powerrail
      Contact( "BA030AZSBK03.00" )
      I_Contact( "Unit1.EmNodes".unitStatus.simulationActive )
   END_RUNG wire#w2
   // the same network as SCL:
   #instcmSuctionPadTopLeftVaccum(enable := TRUE,   // "LBC_TwoWayActuatorCn"
                           parentReferenceDesignator := "Unit1.Em2.Config".em.referenceDesignator.combined,
                           feedbackHomePos := NOT "BA030AZSBK03.00" AND NOT "Unit1.EmNodes".unitStatus.simulationActive,
                           feedbackWorkPos := "BA030AZSBK03.00" AND NOT "Unit1.EmNodes".unitStatus.simulationActive,
                           enableManualCmds := #statEnableManualCmds,
                           interlockWorkPos := "Unit1.Em2.ControlNodes".cm.Interlock.suctionPadTopLeftVaccum.work,
                           interlockHomePos := "Unit1.Em2.ControlNodes".cm.Interlock.suctionPadTopLeftVaccum.home,
                           configuration := "Unit1.Em2.Config".cmSuctionPadTopLeftVaccum,
                           moduleInterface := "Unit1.Em2.HmiInterface".cmSuctionPadTopLeftVaccum,
                           controlNode := "Unit1.Em2.ControlNodes".cmSuctionPadTopLeftVaccum,
                           goToHomePos => "BA030AZSBK29.01",
                           goToWorkPos => "BA030AZSBK29.00");
END_REGION

REGION Network 97: cmSuctionPadTopRightVaccum Interlock
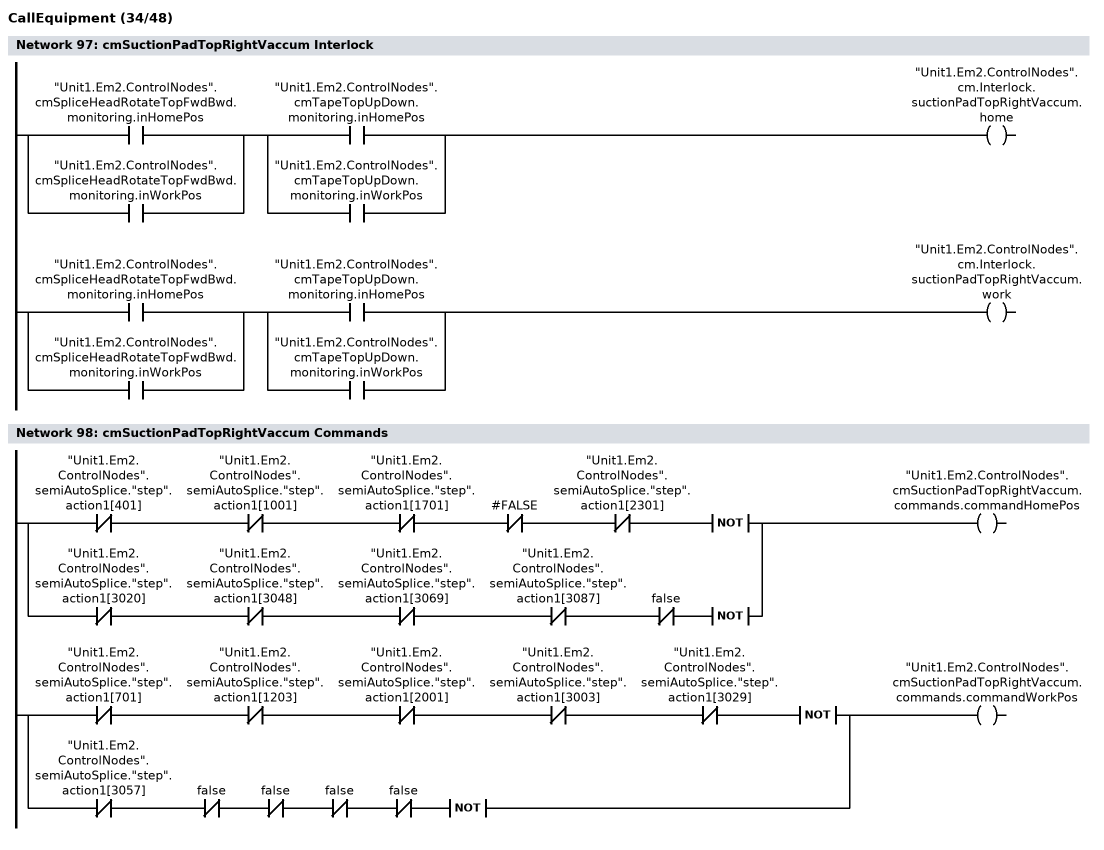
   RUNG wire#powerrail
      Contact( "Unit1.Em2.ControlNodes".cmSpliceHeadRotateTopFwdBwd.monitoring.inHomePos )
      wire#w1
      Contact( "Unit1.Em2.ControlNodes".cmTapeTopUpDown.monitoring.inHomePos )
      wire#w2
      Coil( "Unit1.Em2.ControlNodes".cm.Interlock.suctionPadTopRightVaccum.home )
   END_RUNG
   RUNG wire#powerrail
      Contact( "Unit1.Em2.ControlNodes".cmSpliceHeadRotateTopFwdBwd.monitoring.inWorkPos )
   END_RUNG wire#w1
   RUNG wire#w1
      Contact( "Unit1.Em2.ControlNodes".cmTapeTopUpDown.monitoring.inWorkPos )
   END_RUNG wire#w2
   RUNG wire#powerrail
      Contact( "Unit1.Em2.ControlNodes".cmSpliceHeadRotateTopFwdBwd.monitoring.inHomePos )
      wire#w3
      Contact( "Unit1.Em2.ControlNodes".cmTapeTopUpDown.monitoring.inHomePos )
      wire#w4
      Coil( "Unit1.Em2.ControlNodes".cm.Interlock.suctionPadTopRightVaccum.work )
   END_RUNG
   RUNG wire#powerrail
      Contact( "Unit1.Em2.ControlNodes".cmSpliceHeadRotateTopFwdBwd.monitoring.inWorkPos )
   END_RUNG wire#w3
   RUNG wire#w3
      Contact( "Unit1.Em2.ControlNodes".cmTapeTopUpDown.monitoring.inWorkPos )
   END_RUNG wire#w4
   // the same network as SCL:
   "Unit1.Em2.ControlNodes".cm.Interlock.suctionPadTopRightVaccum.home := ("Unit1.Em2.ControlNodes".cmSpliceHeadRotateTopFwdBwd.monitoring.inHomePos OR "Unit1.Em2.ControlNodes".cmSpliceHeadRotateTopFwdBwd.monitoring.inWorkPos) AND ("Unit1.Em2.ControlNodes".cmTapeTopUpDown.monitoring.inHomePos OR "Unit1.Em2.ControlNodes".cmTapeTopUpDown.monitoring.inWorkPos);
   "Unit1.Em2.ControlNodes".cm.Interlock.suctionPadTopRightVaccum.work := ("Unit1.Em2.ControlNodes".cmSpliceHeadRotateTopFwdBwd.monitoring.inHomePos OR "Unit1.Em2.ControlNodes".cmSpliceHeadRotateTopFwdBwd.monitoring.inWorkPos) AND ("Unit1.Em2.ControlNodes".cmTapeTopUpDown.monitoring.inHomePos OR "Unit1.Em2.ControlNodes".cmTapeTopUpDown.monitoring.inWorkPos);
END_REGION

REGION Network 98: cmSuctionPadTopRightVaccum Commands
   RUNG wire#powerrail
      I_Contact( "Unit1.Em2.ControlNodes".semiAutoSplice."step".action1[401] )
      I_Contact( "Unit1.Em2.ControlNodes".semiAutoSplice."step".action1[1001] )
      I_Contact( "Unit1.Em2.ControlNodes".semiAutoSplice."step".action1[1701] )
      I_Contact( #FALSE )
      I_Contact( "Unit1.Em2.ControlNodes".semiAutoSplice."step".action1[2301] )
      Not()
      wire#w1
      Coil( "Unit1.Em2.ControlNodes".cmSuctionPadTopRightVaccum.commands.commandHomePos )
   END_RUNG
   RUNG wire#powerrail
      I_Contact( "Unit1.Em2.ControlNodes".semiAutoSplice."step".action1[3020] )
      I_Contact( "Unit1.Em2.ControlNodes".semiAutoSplice."step".action1[3048] )
      I_Contact( "Unit1.Em2.ControlNodes".semiAutoSplice."step".action1[3069] )
      I_Contact( "Unit1.Em2.ControlNodes".semiAutoSplice."step".action1[3087] )
      I_Contact( false )
      Not()
   END_RUNG wire#w1
   RUNG wire#powerrail
      I_Contact( "Unit1.Em2.ControlNodes".semiAutoSplice."step".action1[701] )
      I_Contact( "Unit1.Em2.ControlNodes".semiAutoSplice."step".action1[1203] )
      I_Contact( "Unit1.Em2.ControlNodes".semiAutoSplice."step".action1[2001] )
      I_Contact( "Unit1.Em2.ControlNodes".semiAutoSplice."step".action1[3003] )
      I_Contact( "Unit1.Em2.ControlNodes".semiAutoSplice."step".action1[3029] )
      Not()
      wire#w2
      Coil( "Unit1.Em2.ControlNodes".cmSuctionPadTopRightVaccum.commands.commandWorkPos )
   END_RUNG
   RUNG wire#powerrail
      I_Contact( "Unit1.Em2.ControlNodes".semiAutoSplice."step".action1[3057] )
      I_Contact( false )
      I_Contact( false )
      I_Contact( false )
      I_Contact( false )
      Not()
   END_RUNG wire#w2
   // the same network as SCL:
   "Unit1.Em2.ControlNodes".cmSuctionPadTopRightVaccum.commands.commandHomePos := NOT (NOT "Unit1.Em2.ControlNodes".semiAutoSplice."step".action1[401] AND NOT "Unit1.Em2.ControlNodes".semiAutoSplice."step".action1[1001] AND NOT "Unit1.Em2.ControlNodes".semiAutoSplice."step".action1[1701] AND NOT #FALSE AND NOT "Unit1.Em2.ControlNodes".semiAutoSplice."step".action1[2301]) OR NOT (NOT "Unit1.Em2.ControlNodes".semiAutoSplice."step".action1[3020] AND NOT "Unit1.Em2.ControlNodes".semiAutoSplice."step".action1[3048] AND NOT "Unit1.Em2.ControlNodes".semiAutoSplice."step".action1[3069] AND NOT "Unit1.Em2.ControlNodes".semiAutoSplice."step".action1[3087] AND NOT false);
   "Unit1.Em2.ControlNodes".cmSuctionPadTopRightVaccum.commands.commandWorkPos := NOT (NOT "Unit1.Em2.ControlNodes".semiAutoSplice."step".action1[701] AND NOT "Unit1.Em2.ControlNodes".semiAutoSplice."step".action1[1203] AND NOT "Unit1.Em2.ControlNodes".semiAutoSplice."step".action1[2001] AND NOT "Unit1.Em2.ControlNodes".semiAutoSplice."step".action1[3003] AND NOT "Unit1.Em2.ControlNodes".semiAutoSplice."step".action1[3029]) OR NOT (NOT "Unit1.Em2.ControlNodes".semiAutoSplice."step".action1[3057] AND NOT false AND NOT false AND NOT false AND NOT false);
END_REGION

REGION Network 99: Call instcmSuctionPadTopRightVaccum (LBC_TwoWayActuator)
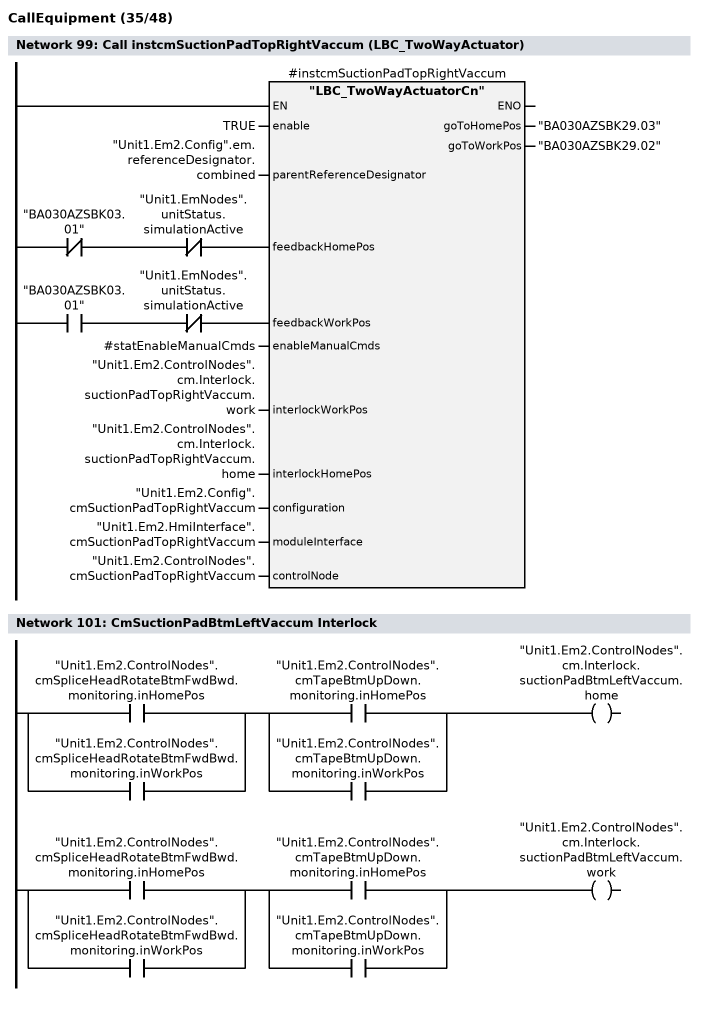
   RUNG wire#powerrail
      #instcmSuctionPadTopRightVaccum(feedbackHomePos := wire#w1, feedbackWorkPos := wire#w2, enable := TRUE, parentReferenceDesignator := "Unit1.Em2.Config".em.referenceDesignator.combined, enableManualCmds := #statEnableManualCmds, interlockWorkPos := "Unit1.Em2.ControlNodes".cm.Interlock.suctionPadTopRightVaccum.work, interlockHomePos := "Unit1.Em2.ControlNodes".cm.Interlock.suctionPadTopRightVaccum.home, configuration := "Unit1.Em2.Config".cmSuctionPadTopRightVaccum, moduleInterface := "Unit1.Em2.HmiInterface".cmSuctionPadTopRightVaccum, controlNode := "Unit1.Em2.ControlNodes".cmSuctionPadTopRightVaccum, goToHomePos => "BA030AZSBK29.03", goToWorkPos => "BA030AZSBK29.02")
   END_RUNG
   RUNG wire#powerrail
      I_Contact( "BA030AZSBK03.01" )
      I_Contact( "Unit1.EmNodes".unitStatus.simulationActive )
   END_RUNG wire#w1
   RUNG wire#powerrail
      Contact( "BA030AZSBK03.01" )
      I_Contact( "Unit1.EmNodes".unitStatus.simulationActive )
   END_RUNG wire#w2
   // the same network as SCL:
   #instcmSuctionPadTopRightVaccum(enable := TRUE,   // "LBC_TwoWayActuatorCn"
                           parentReferenceDesignator := "Unit1.Em2.Config".em.referenceDesignator.combined,
                           feedbackHomePos := NOT "BA030AZSBK03.01" AND NOT "Unit1.EmNodes".unitStatus.simulationActive,
                           feedbackWorkPos := "BA030AZSBK03.01" AND NOT "Unit1.EmNodes".unitStatus.simulationActive,
                           enableManualCmds := #statEnableManualCmds,
                           interlockWorkPos := "Unit1.Em2.ControlNodes".cm.Interlock.suctionPadTopRightVaccum.work,
                           interlockHomePos := "Unit1.Em2.ControlNodes".cm.Interlock.suctionPadTopRightVaccum.home,
                           configuration := "Unit1.Em2.Config".cmSuctionPadTopRightVaccum,
                           moduleInterface := "Unit1.Em2.HmiInterface".cmSuctionPadTopRightVaccum,
                           controlNode := "Unit1.Em2.ControlNodes".cmSuctionPadTopRightVaccum,
                           goToHomePos => "BA030AZSBK29.03",
                           goToWorkPos => "BA030AZSBK29.02");
END_REGION

REGION Network 101: CmSuctionPadBtmLeftVaccum Interlock
   RUNG wire#powerrail
      Contact( "Unit1.Em2.ControlNodes".cmSpliceHeadRotateBtmFwdBwd.monitoring.inHomePos )
      wire#w1
      Contact( "Unit1.Em2.ControlNodes".cmTapeBtmUpDown.monitoring.inHomePos )
      wire#w2
      Coil( "Unit1.Em2.ControlNodes".cm.Interlock.suctionPadBtmLeftVaccum.home )
   END_RUNG
   RUNG wire#powerrail
      Contact( "Unit1.Em2.ControlNodes".cmSpliceHeadRotateBtmFwdBwd.monitoring.inWorkPos )
   END_RUNG wire#w1
   RUNG wire#w1
      Contact( "Unit1.Em2.ControlNodes".cmTapeBtmUpDown.monitoring.inWorkPos )
   END_RUNG wire#w2
   RUNG wire#powerrail
      Contact( "Unit1.Em2.ControlNodes".cmSpliceHeadRotateBtmFwdBwd.monitoring.inHomePos )
      wire#w3
      Contact( "Unit1.Em2.ControlNodes".cmTapeBtmUpDown.monitoring.inHomePos )
      wire#w4
      Coil( "Unit1.Em2.ControlNodes".cm.Interlock.suctionPadBtmLeftVaccum.work )
   END_RUNG
   RUNG wire#powerrail
      Contact( "Unit1.Em2.ControlNodes".cmSpliceHeadRotateBtmFwdBwd.monitoring.inWorkPos )
   END_RUNG wire#w3
   RUNG wire#w3
      Contact( "Unit1.Em2.ControlNodes".cmTapeBtmUpDown.monitoring.inWorkPos )
   END_RUNG wire#w4
   // the same network as SCL:
   "Unit1.Em2.ControlNodes".cm.Interlock.suctionPadBtmLeftVaccum.home := ("Unit1.Em2.ControlNodes".cmSpliceHeadRotateBtmFwdBwd.monitoring.inHomePos OR "Unit1.Em2.ControlNodes".cmSpliceHeadRotateBtmFwdBwd.monitoring.inWorkPos) AND ("Unit1.Em2.ControlNodes".cmTapeBtmUpDown.monitoring.inHomePos OR "Unit1.Em2.ControlNodes".cmTapeBtmUpDown.monitoring.inWorkPos);
   "Unit1.Em2.ControlNodes".cm.Interlock.suctionPadBtmLeftVaccum.work := ("Unit1.Em2.ControlNodes".cmSpliceHeadRotateBtmFwdBwd.monitoring.inHomePos OR "Unit1.Em2.ControlNodes".cmSpliceHeadRotateBtmFwdBwd.monitoring.inWorkPos) AND ("Unit1.Em2.ControlNodes".cmTapeBtmUpDown.monitoring.inHomePos OR "Unit1.Em2.ControlNodes".cmTapeBtmUpDown.monitoring.inWorkPos);
END_REGION

REGION Network 102: CmSuctionPadBtmLeftVaccum Commands
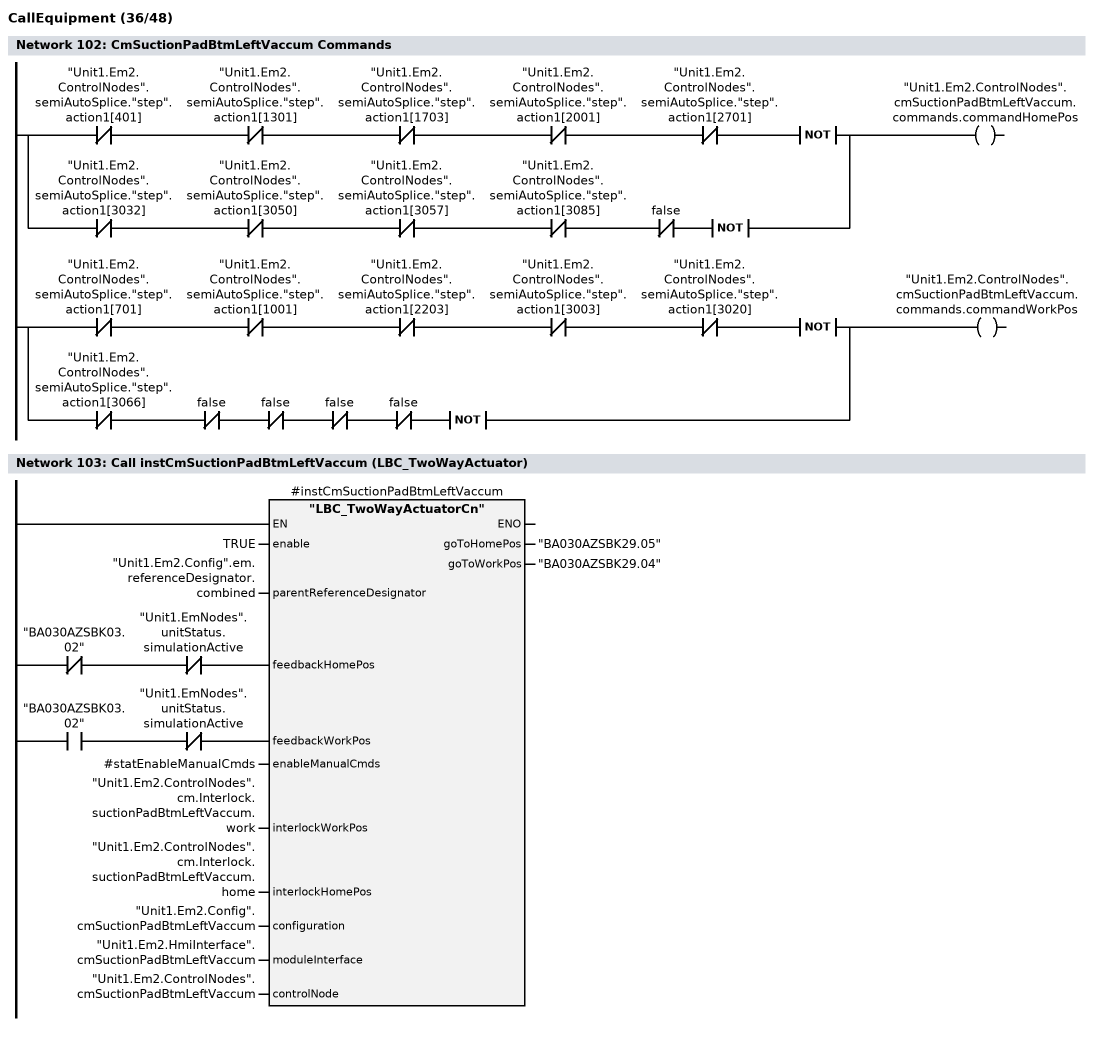
   RUNG wire#powerrail
      I_Contact( "Unit1.Em2.ControlNodes".semiAutoSplice."step".action1[401] )
      I_Contact( "Unit1.Em2.ControlNodes".semiAutoSplice."step".action1[1301] )
      I_Contact( "Unit1.Em2.ControlNodes".semiAutoSplice."step".action1[1703] )
      I_Contact( "Unit1.Em2.ControlNodes".semiAutoSplice."step".action1[2001] )
      I_Contact( "Unit1.Em2.ControlNodes".semiAutoSplice."step".action1[2701] )
      Not()
      wire#w1
      Coil( "Unit1.Em2.ControlNodes".cmSuctionPadBtmLeftVaccum.commands.commandHomePos )
   END_RUNG
   RUNG wire#powerrail
      I_Contact( "Unit1.Em2.ControlNodes".semiAutoSplice."step".action1[3032] )
      I_Contact( "Unit1.Em2.ControlNodes".semiAutoSplice."step".action1[3050] )
      I_Contact( "Unit1.Em2.ControlNodes".semiAutoSplice."step".action1[3057] )
      I_Contact( "Unit1.Em2.ControlNodes".semiAutoSplice."step".action1[3085] )
      I_Contact( false )
      Not()
   END_RUNG wire#w1
   RUNG wire#powerrail
      I_Contact( "Unit1.Em2.ControlNodes".semiAutoSplice."step".action1[701] )
      I_Contact( "Unit1.Em2.ControlNodes".semiAutoSplice."step".action1[1001] )
      I_Contact( "Unit1.Em2.ControlNodes".semiAutoSplice."step".action1[2203] )
      I_Contact( "Unit1.Em2.ControlNodes".semiAutoSplice."step".action1[3003] )
      I_Contact( "Unit1.Em2.ControlNodes".semiAutoSplice."step".action1[3020] )
      Not()
      wire#w2
      Coil( "Unit1.Em2.ControlNodes".cmSuctionPadBtmLeftVaccum.commands.commandWorkPos )
   END_RUNG
   RUNG wire#powerrail
      I_Contact( "Unit1.Em2.ControlNodes".semiAutoSplice."step".action1[3066] )
      I_Contact( false )
      I_Contact( false )
      I_Contact( false )
      I_Contact( false )
      Not()
   END_RUNG wire#w2
   // the same network as SCL:
   "Unit1.Em2.ControlNodes".cmSuctionPadBtmLeftVaccum.commands.commandHomePos := NOT (NOT "Unit1.Em2.ControlNodes".semiAutoSplice."step".action1[401] AND NOT "Unit1.Em2.ControlNodes".semiAutoSplice."step".action1[1301] AND NOT "Unit1.Em2.ControlNodes".semiAutoSplice."step".action1[1703] AND NOT "Unit1.Em2.ControlNodes".semiAutoSplice."step".action1[2001] AND NOT "Unit1.Em2.ControlNodes".semiAutoSplice."step".action1[2701]) OR NOT (NOT "Unit1.Em2.ControlNodes".semiAutoSplice."step".action1[3032] AND NOT "Unit1.Em2.ControlNodes".semiAutoSplice."step".action1[3050] AND NOT "Unit1.Em2.ControlNodes".semiAutoSplice."step".action1[3057] AND NOT "Unit1.Em2.ControlNodes".semiAutoSplice."step".action1[3085] AND NOT false);
   "Unit1.Em2.ControlNodes".cmSuctionPadBtmLeftVaccum.commands.commandWorkPos := NOT (NOT "Unit1.Em2.ControlNodes".semiAutoSplice."step".action1[701] AND NOT "Unit1.Em2.ControlNodes".semiAutoSplice."step".action1[1001] AND NOT "Unit1.Em2.ControlNodes".semiAutoSplice."step".action1[2203] AND NOT "Unit1.Em2.ControlNodes".semiAutoSplice."step".action1[3003] AND NOT "Unit1.Em2.ControlNodes".semiAutoSplice."step".action1[3020]) OR NOT (NOT "Unit1.Em2.ControlNodes".semiAutoSplice."step".action1[3066] AND NOT false AND NOT false AND NOT false AND NOT false);
END_REGION

REGION Network 103: Call instCmSuctionPadBtmLeftVaccum (LBC_TwoWayActuator)
   RUNG wire#powerrail
      #instCmSuctionPadBtmLeftVaccum(feedbackHomePos := wire#w1, feedbackWorkPos := wire#w2, enable := TRUE, parentReferenceDesignator := "Unit1.Em2.Config".em.referenceDesignator.combined, enableManualCmds := #statEnableManualCmds, interlockWorkPos := "Unit1.Em2.ControlNodes".cm.Interlock.suctionPadBtmLeftVaccum.work, interlockHomePos := "Unit1.Em2.ControlNodes".cm.Interlock.suctionPadBtmLeftVaccum.home, configuration := "Unit1.Em2.Config".cmSuctionPadBtmLeftVaccum, moduleInterface := "Unit1.Em2.HmiInterface".cmSuctionPadBtmLeftVaccum, controlNode := "Unit1.Em2.ControlNodes".cmSuctionPadBtmLeftVaccum, goToHomePos => "BA030AZSBK29.05", goToWorkPos => "BA030AZSBK29.04")
   END_RUNG
   RUNG wire#powerrail
      I_Contact( "BA030AZSBK03.02" )
      I_Contact( "Unit1.EmNodes".unitStatus.simulationActive )
   END_RUNG wire#w1
   RUNG wire#powerrail
      Contact( "BA030AZSBK03.02" )
      I_Contact( "Unit1.EmNodes".unitStatus.simulationActive )
   END_RUNG wire#w2
   // the same network as SCL:
   #instCmSuctionPadBtmLeftVaccum(enable := TRUE,   // "LBC_TwoWayActuatorCn"
                           parentReferenceDesignator := "Unit1.Em2.Config".em.referenceDesignator.combined,
                           feedbackHomePos := NOT "BA030AZSBK03.02" AND NOT "Unit1.EmNodes".unitStatus.simulationActive,
                           feedbackWorkPos := "BA030AZSBK03.02" AND NOT "Unit1.EmNodes".unitStatus.simulationActive,
                           enableManualCmds := #statEnableManualCmds,
                           interlockWorkPos := "Unit1.Em2.ControlNodes".cm.Interlock.suctionPadBtmLeftVaccum.work,
                           interlockHomePos := "Unit1.Em2.ControlNodes".cm.Interlock.suctionPadBtmLeftVaccum.home,
                           configuration := "Unit1.Em2.Config".cmSuctionPadBtmLeftVaccum,
                           moduleInterface := "Unit1.Em2.HmiInterface".cmSuctionPadBtmLeftVaccum,
                           controlNode := "Unit1.Em2.ControlNodes".cmSuctionPadBtmLeftVaccum,
                           goToHomePos => "BA030AZSBK29.05",
                           goToWorkPos => "BA030AZSBK29.04");
END_REGION

REGION Network 105: CmSuctionPadBtmRightVaccum Interlock
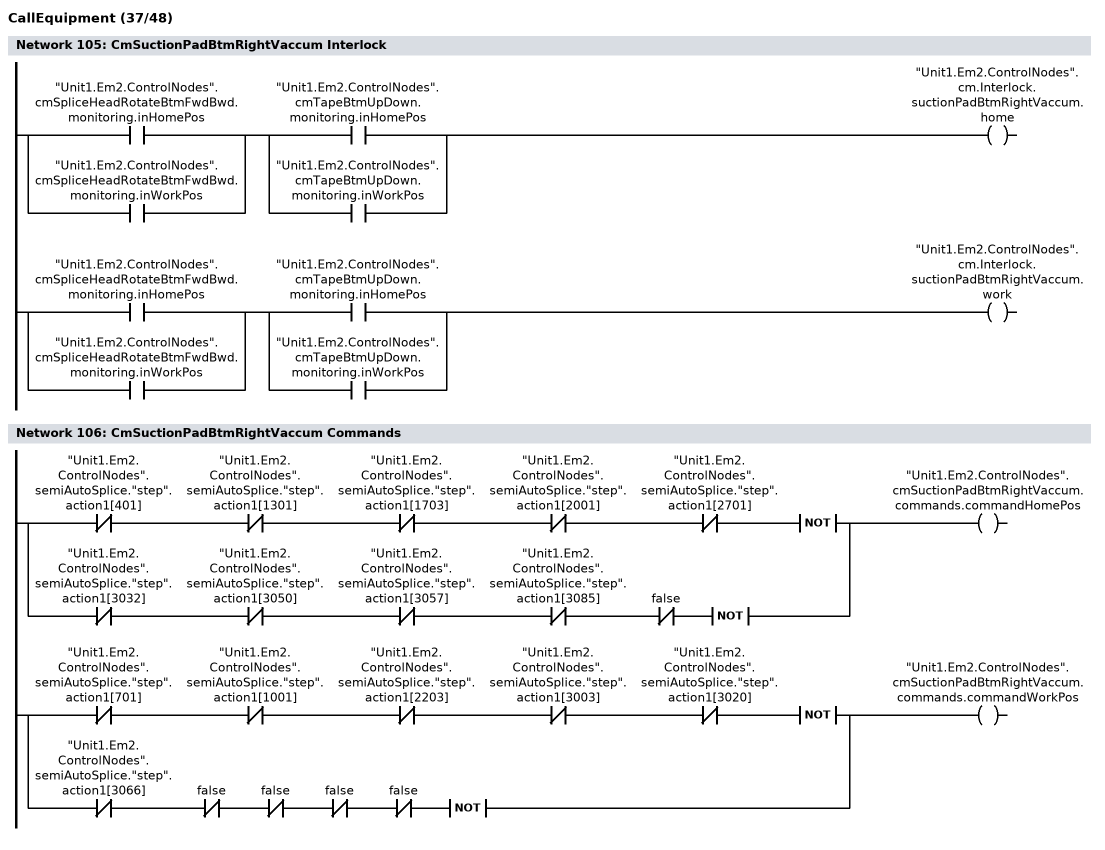
   RUNG wire#powerrail
      Contact( "Unit1.Em2.ControlNodes".cmSpliceHeadRotateBtmFwdBwd.monitoring.inHomePos )
      wire#w1
      Contact( "Unit1.Em2.ControlNodes".cmTapeBtmUpDown.monitoring.inHomePos )
      wire#w2
      Coil( "Unit1.Em2.ControlNodes".cm.Interlock.suctionPadBtmRightVaccum.home )
   END_RUNG
   RUNG wire#powerrail
      Contact( "Unit1.Em2.ControlNodes".cmSpliceHeadRotateBtmFwdBwd.monitoring.inWorkPos )
   END_RUNG wire#w1
   RUNG wire#w1
      Contact( "Unit1.Em2.ControlNodes".cmTapeBtmUpDown.monitoring.inWorkPos )
   END_RUNG wire#w2
   RUNG wire#powerrail
      Contact( "Unit1.Em2.ControlNodes".cmSpliceHeadRotateBtmFwdBwd.monitoring.inHomePos )
      wire#w3
      Contact( "Unit1.Em2.ControlNodes".cmTapeBtmUpDown.monitoring.inHomePos )
      wire#w4
      Coil( "Unit1.Em2.ControlNodes".cm.Interlock.suctionPadBtmRightVaccum.work )
   END_RUNG
   RUNG wire#powerrail
      Contact( "Unit1.Em2.ControlNodes".cmSpliceHeadRotateBtmFwdBwd.monitoring.inWorkPos )
   END_RUNG wire#w3
   RUNG wire#w3
      Contact( "Unit1.Em2.ControlNodes".cmTapeBtmUpDown.monitoring.inWorkPos )
   END_RUNG wire#w4
   // the same network as SCL:
   "Unit1.Em2.ControlNodes".cm.Interlock.suctionPadBtmRightVaccum.home := ("Unit1.Em2.ControlNodes".cmSpliceHeadRotateBtmFwdBwd.monitoring.inHomePos OR "Unit1.Em2.ControlNodes".cmSpliceHeadRotateBtmFwdBwd.monitoring.inWorkPos) AND ("Unit1.Em2.ControlNodes".cmTapeBtmUpDown.monitoring.inHomePos OR "Unit1.Em2.ControlNodes".cmTapeBtmUpDown.monitoring.inWorkPos);
   "Unit1.Em2.ControlNodes".cm.Interlock.suctionPadBtmRightVaccum.work := ("Unit1.Em2.ControlNodes".cmSpliceHeadRotateBtmFwdBwd.monitoring.inHomePos OR "Unit1.Em2.ControlNodes".cmSpliceHeadRotateBtmFwdBwd.monitoring.inWorkPos) AND ("Unit1.Em2.ControlNodes".cmTapeBtmUpDown.monitoring.inHomePos OR "Unit1.Em2.ControlNodes".cmTapeBtmUpDown.monitoring.inWorkPos);
END_REGION

REGION Network 106: CmSuctionPadBtmRightVaccum Commands
   RUNG wire#powerrail
      I_Contact( "Unit1.Em2.ControlNodes".semiAutoSplice."step".action1[401] )
      I_Contact( "Unit1.Em2.ControlNodes".semiAutoSplice."step".action1[1301] )
      I_Contact( "Unit1.Em2.ControlNodes".semiAutoSplice."step".action1[1703] )
      I_Contact( "Unit1.Em2.ControlNodes".semiAutoSplice."step".action1[2001] )
      I_Contact( "Unit1.Em2.ControlNodes".semiAutoSplice."step".action1[2701] )
      Not()
      wire#w1
      Coil( "Unit1.Em2.ControlNodes".cmSuctionPadBtmRightVaccum.commands.commandHomePos )
   END_RUNG
   RUNG wire#powerrail
      I_Contact( "Unit1.Em2.ControlNodes".semiAutoSplice."step".action1[3032] )
      I_Contact( "Unit1.Em2.ControlNodes".semiAutoSplice."step".action1[3050] )
      I_Contact( "Unit1.Em2.ControlNodes".semiAutoSplice."step".action1[3057] )
      I_Contact( "Unit1.Em2.ControlNodes".semiAutoSplice."step".action1[3085] )
      I_Contact( false )
      Not()
   END_RUNG wire#w1
   RUNG wire#powerrail
      I_Contact( "Unit1.Em2.ControlNodes".semiAutoSplice."step".action1[701] )
      I_Contact( "Unit1.Em2.ControlNodes".semiAutoSplice."step".action1[1001] )
      I_Contact( "Unit1.Em2.ControlNodes".semiAutoSplice."step".action1[2203] )
      I_Contact( "Unit1.Em2.ControlNodes".semiAutoSplice."step".action1[3003] )
      I_Contact( "Unit1.Em2.ControlNodes".semiAutoSplice."step".action1[3020] )
      Not()
      wire#w2
      Coil( "Unit1.Em2.ControlNodes".cmSuctionPadBtmRightVaccum.commands.commandWorkPos )
   END_RUNG
   RUNG wire#powerrail
      I_Contact( "Unit1.Em2.ControlNodes".semiAutoSplice."step".action1[3066] )
      I_Contact( false )
      I_Contact( false )
      I_Contact( false )
      I_Contact( false )
      Not()
   END_RUNG wire#w2
   // the same network as SCL:
   "Unit1.Em2.ControlNodes".cmSuctionPadBtmRightVaccum.commands.commandHomePos := NOT (NOT "Unit1.Em2.ControlNodes".semiAutoSplice."step".action1[401] AND NOT "Unit1.Em2.ControlNodes".semiAutoSplice."step".action1[1301] AND NOT "Unit1.Em2.ControlNodes".semiAutoSplice."step".action1[1703] AND NOT "Unit1.Em2.ControlNodes".semiAutoSplice."step".action1[2001] AND NOT "Unit1.Em2.ControlNodes".semiAutoSplice."step".action1[2701]) OR NOT (NOT "Unit1.Em2.ControlNodes".semiAutoSplice."step".action1[3032] AND NOT "Unit1.Em2.ControlNodes".semiAutoSplice."step".action1[3050] AND NOT "Unit1.Em2.ControlNodes".semiAutoSplice."step".action1[3057] AND NOT "Unit1.Em2.ControlNodes".semiAutoSplice."step".action1[3085] AND NOT false);
   "Unit1.Em2.ControlNodes".cmSuctionPadBtmRightVaccum.commands.commandWorkPos := NOT (NOT "Unit1.Em2.ControlNodes".semiAutoSplice."step".action1[701] AND NOT "Unit1.Em2.ControlNodes".semiAutoSplice."step".action1[1001] AND NOT "Unit1.Em2.ControlNodes".semiAutoSplice."step".action1[2203] AND NOT "Unit1.Em2.ControlNodes".semiAutoSplice."step".action1[3003] AND NOT "Unit1.Em2.ControlNodes".semiAutoSplice."step".action1[3020]) OR NOT (NOT "Unit1.Em2.ControlNodes".semiAutoSplice."step".action1[3066] AND NOT false AND NOT false AND NOT false AND NOT false);
END_REGION

REGION Network 107: Call instCmSuctionPadBtmRightVaccum (LBC_TwoWayActuator)
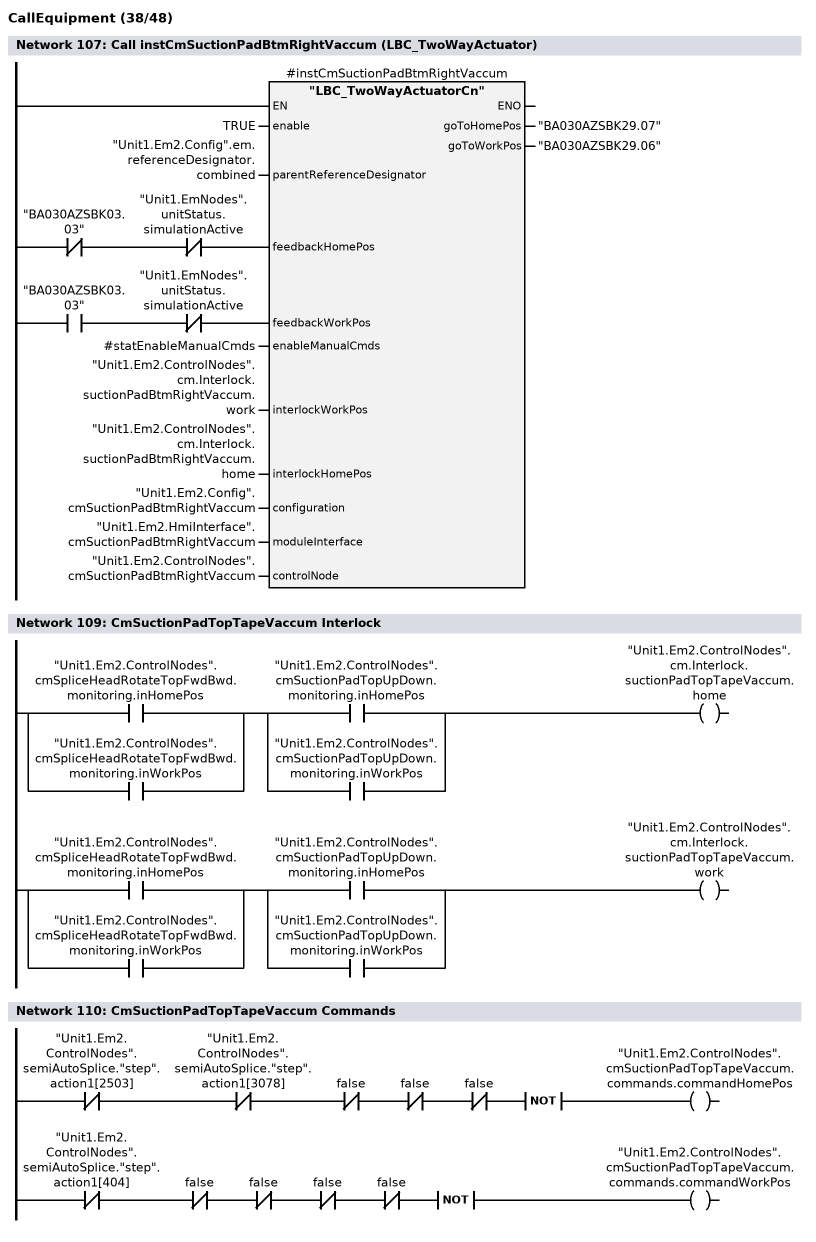
   RUNG wire#powerrail
      #instCmSuctionPadBtmRightVaccum(feedbackHomePos := wire#w1, feedbackWorkPos := wire#w2, enable := TRUE, parentReferenceDesignator := "Unit1.Em2.Config".em.referenceDesignator.combined, enableManualCmds := #statEnableManualCmds, interlockWorkPos := "Unit1.Em2.ControlNodes".cm.Interlock.suctionPadBtmRightVaccum.work, interlockHomePos := "Unit1.Em2.ControlNodes".cm.Interlock.suctionPadBtmRightVaccum.home, configuration := "Unit1.Em2.Config".cmSuctionPadBtmRightVaccum, moduleInterface := "Unit1.Em2.HmiInterface".cmSuctionPadBtmRightVaccum, controlNode := "Unit1.Em2.ControlNodes".cmSuctionPadBtmRightVaccum, goToHomePos => "BA030AZSBK29.07", goToWorkPos => "BA030AZSBK29.06")
   END_RUNG
   RUNG wire#powerrail
      I_Contact( "BA030AZSBK03.03" )
      I_Contact( "Unit1.EmNodes".unitStatus.simulationActive )
   END_RUNG wire#w1
   RUNG wire#powerrail
      Contact( "BA030AZSBK03.03" )
      I_Contact( "Unit1.EmNodes".unitStatus.simulationActive )
   END_RUNG wire#w2
   // the same network as SCL:
   #instCmSuctionPadBtmRightVaccum(enable := TRUE,   // "LBC_TwoWayActuatorCn"
                           parentReferenceDesignator := "Unit1.Em2.Config".em.referenceDesignator.combined,
                           feedbackHomePos := NOT "BA030AZSBK03.03" AND NOT "Unit1.EmNodes".unitStatus.simulationActive,
                           feedbackWorkPos := "BA030AZSBK03.03" AND NOT "Unit1.EmNodes".unitStatus.simulationActive,
                           enableManualCmds := #statEnableManualCmds,
                           interlockWorkPos := "Unit1.Em2.ControlNodes".cm.Interlock.suctionPadBtmRightVaccum.work,
                           interlockHomePos := "Unit1.Em2.ControlNodes".cm.Interlock.suctionPadBtmRightVaccum.home,
                           configuration := "Unit1.Em2.Config".cmSuctionPadBtmRightVaccum,
                           moduleInterface := "Unit1.Em2.HmiInterface".cmSuctionPadBtmRightVaccum,
                           controlNode := "Unit1.Em2.ControlNodes".cmSuctionPadBtmRightVaccum,
                           goToHomePos => "BA030AZSBK29.07",
                           goToWorkPos => "BA030AZSBK29.06");
END_REGION

REGION Network 109: CmSuctionPadTopTapeVaccum Interlock
   RUNG wire#powerrail
      Contact( "Unit1.Em2.ControlNodes".cmSpliceHeadRotateTopFwdBwd.monitoring.inHomePos )
      wire#w1
      Contact( "Unit1.Em2.ControlNodes".cmSuctionPadTopUpDown.monitoring.inHomePos )
      wire#w2
      Coil( "Unit1.Em2.ControlNodes".cm.Interlock.suctionPadTopTapeVaccum.home )
   END_RUNG
   RUNG wire#powerrail
      Contact( "Unit1.Em2.ControlNodes".cmSpliceHeadRotateTopFwdBwd.monitoring.inWorkPos )
   END_RUNG wire#w1
   RUNG wire#w1
      Contact( "Unit1.Em2.ControlNodes".cmSuctionPadTopUpDown.monitoring.inWorkPos )
   END_RUNG wire#w2
   RUNG wire#powerrail
      Contact( "Unit1.Em2.ControlNodes".cmSpliceHeadRotateTopFwdBwd.monitoring.inHomePos )
      wire#w3
      Contact( "Unit1.Em2.ControlNodes".cmSuctionPadTopUpDown.monitoring.inHomePos )
      wire#w4
      Coil( "Unit1.Em2.ControlNodes".cm.Interlock.suctionPadTopTapeVaccum.work )
   END_RUNG
   RUNG wire#powerrail
      Contact( "Unit1.Em2.ControlNodes".cmSpliceHeadRotateTopFwdBwd.monitoring.inWorkPos )
   END_RUNG wire#w3
   RUNG wire#w3
      Contact( "Unit1.Em2.ControlNodes".cmSuctionPadTopUpDown.monitoring.inWorkPos )
   END_RUNG wire#w4
   // the same network as SCL:
   "Unit1.Em2.ControlNodes".cm.Interlock.suctionPadTopTapeVaccum.home := ("Unit1.Em2.ControlNodes".cmSpliceHeadRotateTopFwdBwd.monitoring.inHomePos OR "Unit1.Em2.ControlNodes".cmSpliceHeadRotateTopFwdBwd.monitoring.inWorkPos) AND ("Unit1.Em2.ControlNodes".cmSuctionPadTopUpDown.monitoring.inHomePos OR "Unit1.Em2.ControlNodes".cmSuctionPadTopUpDown.monitoring.inWorkPos);
   "Unit1.Em2.ControlNodes".cm.Interlock.suctionPadTopTapeVaccum.work := ("Unit1.Em2.ControlNodes".cmSpliceHeadRotateTopFwdBwd.monitoring.inHomePos OR "Unit1.Em2.ControlNodes".cmSpliceHeadRotateTopFwdBwd.monitoring.inWorkPos) AND ("Unit1.Em2.ControlNodes".cmSuctionPadTopUpDown.monitoring.inHomePos OR "Unit1.Em2.ControlNodes".cmSuctionPadTopUpDown.monitoring.inWorkPos);
END_REGION

REGION Network 110: CmSuctionPadTopTapeVaccum Commands
   RUNG wire#powerrail
      I_Contact( "Unit1.Em2.ControlNodes".semiAutoSplice."step".action1[2503] )
      I_Contact( "Unit1.Em2.ControlNodes".semiAutoSplice."step".action1[3078] )
      I_Contact( false )
      I_Contact( false )
      I_Contact( false )
      Not()
      Coil( "Unit1.Em2.ControlNodes".cmSuctionPadTopTapeVaccum.commands.commandHomePos )
   END_RUNG
   RUNG wire#powerrail
      I_Contact( "Unit1.Em2.ControlNodes".semiAutoSplice."step".action1[404] )
      I_Contact( false )
      I_Contact( false )
      I_Contact( false )
      I_Contact( false )
      Not()
      Coil( "Unit1.Em2.ControlNodes".cmSuctionPadTopTapeVaccum.commands.commandWorkPos )
   END_RUNG
   // the same network as SCL:
   "Unit1.Em2.ControlNodes".cmSuctionPadTopTapeVaccum.commands.commandHomePos := NOT (NOT "Unit1.Em2.ControlNodes".semiAutoSplice."step".action1[2503] AND NOT "Unit1.Em2.ControlNodes".semiAutoSplice."step".action1[3078] AND NOT false AND NOT false AND NOT false);
   "Unit1.Em2.ControlNodes".cmSuctionPadTopTapeVaccum.commands.commandWorkPos := NOT (NOT "Unit1.Em2.ControlNodes".semiAutoSplice."step".action1[404] AND NOT false AND NOT false AND NOT false AND NOT false);
END_REGION

REGION Network 111: Call instCmSuctionPadTopTapeVaccum (LBC_TwoWayActuator)
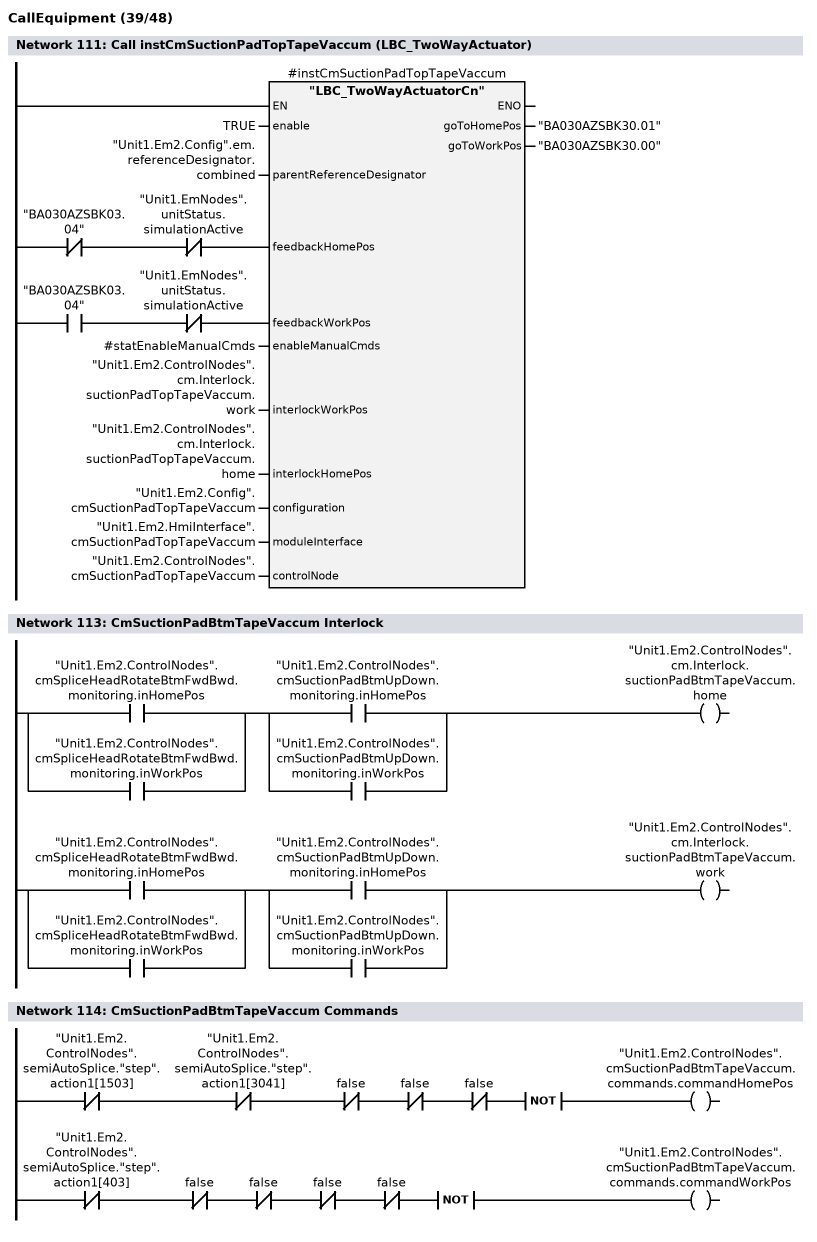
   RUNG wire#powerrail
      #instCmSuctionPadTopTapeVaccum(feedbackHomePos := wire#w1, feedbackWorkPos := wire#w2, enable := TRUE, parentReferenceDesignator := "Unit1.Em2.Config".em.referenceDesignator.combined, enableManualCmds := #statEnableManualCmds, interlockWorkPos := "Unit1.Em2.ControlNodes".cm.Interlock.suctionPadTopTapeVaccum.work, interlockHomePos := "Unit1.Em2.ControlNodes".cm.Interlock.suctionPadTopTapeVaccum.home, configuration := "Unit1.Em2.Config".cmSuctionPadTopTapeVaccum, moduleInterface := "Unit1.Em2.HmiInterface".cmSuctionPadTopTapeVaccum, controlNode := "Unit1.Em2.ControlNodes".cmSuctionPadTopTapeVaccum, goToHomePos => "BA030AZSBK30.01", goToWorkPos => "BA030AZSBK30.00")
   END_RUNG
   RUNG wire#powerrail
      I_Contact( "BA030AZSBK03.04" )
      I_Contact( "Unit1.EmNodes".unitStatus.simulationActive )
   END_RUNG wire#w1
   RUNG wire#powerrail
      Contact( "BA030AZSBK03.04" )
      I_Contact( "Unit1.EmNodes".unitStatus.simulationActive )
   END_RUNG wire#w2
   // the same network as SCL:
   #instCmSuctionPadTopTapeVaccum(enable := TRUE,   // "LBC_TwoWayActuatorCn"
                           parentReferenceDesignator := "Unit1.Em2.Config".em.referenceDesignator.combined,
                           feedbackHomePos := NOT "BA030AZSBK03.04" AND NOT "Unit1.EmNodes".unitStatus.simulationActive,
                           feedbackWorkPos := "BA030AZSBK03.04" AND NOT "Unit1.EmNodes".unitStatus.simulationActive,
                           enableManualCmds := #statEnableManualCmds,
                           interlockWorkPos := "Unit1.Em2.ControlNodes".cm.Interlock.suctionPadTopTapeVaccum.work,
                           interlockHomePos := "Unit1.Em2.ControlNodes".cm.Interlock.suctionPadTopTapeVaccum.home,
                           configuration := "Unit1.Em2.Config".cmSuctionPadTopTapeVaccum,
                           moduleInterface := "Unit1.Em2.HmiInterface".cmSuctionPadTopTapeVaccum,
                           controlNode := "Unit1.Em2.ControlNodes".cmSuctionPadTopTapeVaccum,
                           goToHomePos => "BA030AZSBK30.01",
                           goToWorkPos => "BA030AZSBK30.00");
END_REGION

REGION Network 113: CmSuctionPadBtmTapeVaccum Interlock
   RUNG wire#powerrail
      Contact( "Unit1.Em2.ControlNodes".cmSpliceHeadRotateBtmFwdBwd.monitoring.inHomePos )
      wire#w1
      Contact( "Unit1.Em2.ControlNodes".cmSuctionPadBtmUpDown.monitoring.inHomePos )
      wire#w2
      Coil( "Unit1.Em2.ControlNodes".cm.Interlock.suctionPadBtmTapeVaccum.home )
   END_RUNG
   RUNG wire#powerrail
      Contact( "Unit1.Em2.ControlNodes".cmSpliceHeadRotateBtmFwdBwd.monitoring.inWorkPos )
   END_RUNG wire#w1
   RUNG wire#w1
      Contact( "Unit1.Em2.ControlNodes".cmSuctionPadBtmUpDown.monitoring.inWorkPos )
   END_RUNG wire#w2
   RUNG wire#powerrail
      Contact( "Unit1.Em2.ControlNodes".cmSpliceHeadRotateBtmFwdBwd.monitoring.inHomePos )
      wire#w3
      Contact( "Unit1.Em2.ControlNodes".cmSuctionPadBtmUpDown.monitoring.inHomePos )
      wire#w4
      Coil( "Unit1.Em2.ControlNodes".cm.Interlock.suctionPadBtmTapeVaccum.work )
   END_RUNG
   RUNG wire#powerrail
      Contact( "Unit1.Em2.ControlNodes".cmSpliceHeadRotateBtmFwdBwd.monitoring.inWorkPos )
   END_RUNG wire#w3
   RUNG wire#w3
      Contact( "Unit1.Em2.ControlNodes".cmSuctionPadBtmUpDown.monitoring.inWorkPos )
   END_RUNG wire#w4
   // the same network as SCL:
   "Unit1.Em2.ControlNodes".cm.Interlock.suctionPadBtmTapeVaccum.home := ("Unit1.Em2.ControlNodes".cmSpliceHeadRotateBtmFwdBwd.monitoring.inHomePos OR "Unit1.Em2.ControlNodes".cmSpliceHeadRotateBtmFwdBwd.monitoring.inWorkPos) AND ("Unit1.Em2.ControlNodes".cmSuctionPadBtmUpDown.monitoring.inHomePos OR "Unit1.Em2.ControlNodes".cmSuctionPadBtmUpDown.monitoring.inWorkPos);
   "Unit1.Em2.ControlNodes".cm.Interlock.suctionPadBtmTapeVaccum.work := ("Unit1.Em2.ControlNodes".cmSpliceHeadRotateBtmFwdBwd.monitoring.inHomePos OR "Unit1.Em2.ControlNodes".cmSpliceHeadRotateBtmFwdBwd.monitoring.inWorkPos) AND ("Unit1.Em2.ControlNodes".cmSuctionPadBtmUpDown.monitoring.inHomePos OR "Unit1.Em2.ControlNodes".cmSuctionPadBtmUpDown.monitoring.inWorkPos);
END_REGION

REGION Network 114: CmSuctionPadBtmTapeVaccum Commands
   RUNG wire#powerrail
      I_Contact( "Unit1.Em2.ControlNodes".semiAutoSplice."step".action1[1503] )
      I_Contact( "Unit1.Em2.ControlNodes".semiAutoSplice."step".action1[3041] )
      I_Contact( false )
      I_Contact( false )
      I_Contact( false )
      Not()
      Coil( "Unit1.Em2.ControlNodes".cmSuctionPadBtmTapeVaccum.commands.commandHomePos )
   END_RUNG
   RUNG wire#powerrail
      I_Contact( "Unit1.Em2.ControlNodes".semiAutoSplice."step".action1[403] )
      I_Contact( false )
      I_Contact( false )
      I_Contact( false )
      I_Contact( false )
      Not()
      Coil( "Unit1.Em2.ControlNodes".cmSuctionPadBtmTapeVaccum.commands.commandWorkPos )
   END_RUNG
   // the same network as SCL:
   "Unit1.Em2.ControlNodes".cmSuctionPadBtmTapeVaccum.commands.commandHomePos := NOT (NOT "Unit1.Em2.ControlNodes".semiAutoSplice."step".action1[1503] AND NOT "Unit1.Em2.ControlNodes".semiAutoSplice."step".action1[3041] AND NOT false AND NOT false AND NOT false);
   "Unit1.Em2.ControlNodes".cmSuctionPadBtmTapeVaccum.commands.commandWorkPos := NOT (NOT "Unit1.Em2.ControlNodes".semiAutoSplice."step".action1[403] AND NOT false AND NOT false AND NOT false AND NOT false);
END_REGION

REGION Network 115: Call instCmSuctionPadBtmTapeVaccum (LBC_TwoWayActuator)
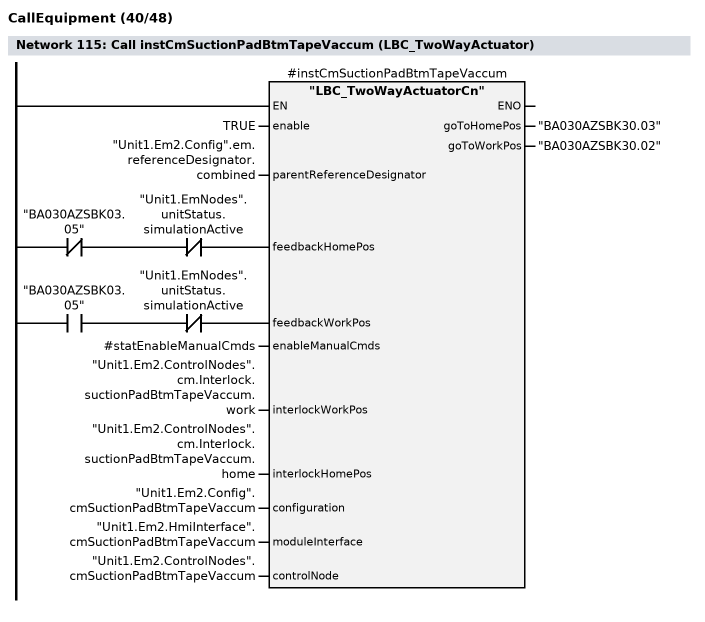
   RUNG wire#powerrail
      #instCmSuctionPadBtmTapeVaccum(feedbackHomePos := wire#w1, feedbackWorkPos := wire#w2, enable := TRUE, parentReferenceDesignator := "Unit1.Em2.Config".em.referenceDesignator.combined, enableManualCmds := #statEnableManualCmds, interlockWorkPos := "Unit1.Em2.ControlNodes".cm.Interlock.suctionPadBtmTapeVaccum.work, interlockHomePos := "Unit1.Em2.ControlNodes".cm.Interlock.suctionPadBtmTapeVaccum.home, configuration := "Unit1.Em2.Config".cmSuctionPadBtmTapeVaccum, moduleInterface := "Unit1.Em2.HmiInterface".cmSuctionPadBtmTapeVaccum, controlNode := "Unit1.Em2.ControlNodes".cmSuctionPadBtmTapeVaccum, goToHomePos => "BA030AZSBK30.03", goToWorkPos => "BA030AZSBK30.02")
   END_RUNG
   RUNG wire#powerrail
      I_Contact( "BA030AZSBK03.05" )
      I_Contact( "Unit1.EmNodes".unitStatus.simulationActive )
   END_RUNG wire#w1
   RUNG wire#powerrail
      Contact( "BA030AZSBK03.05" )
      I_Contact( "Unit1.EmNodes".unitStatus.simulationActive )
   END_RUNG wire#w2
   // the same network as SCL:
   #instCmSuctionPadBtmTapeVaccum(enable := TRUE,   // "LBC_TwoWayActuatorCn"
                           parentReferenceDesignator := "Unit1.Em2.Config".em.referenceDesignator.combined,
                           feedbackHomePos := NOT "BA030AZSBK03.05" AND NOT "Unit1.EmNodes".unitStatus.simulationActive,
                           feedbackWorkPos := "BA030AZSBK03.05" AND NOT "Unit1.EmNodes".unitStatus.simulationActive,
                           enableManualCmds := #statEnableManualCmds,
                           interlockWorkPos := "Unit1.Em2.ControlNodes".cm.Interlock.suctionPadBtmTapeVaccum.work,
                           interlockHomePos := "Unit1.Em2.ControlNodes".cm.Interlock.suctionPadBtmTapeVaccum.home,
                           configuration := "Unit1.Em2.Config".cmSuctionPadBtmTapeVaccum,
                           moduleInterface := "Unit1.Em2.HmiInterface".cmSuctionPadBtmTapeVaccum,
                           controlNode := "Unit1.Em2.ControlNodes".cmSuctionPadBtmTapeVaccum,
                           goToHomePos => "BA030AZSBK30.03",
                           goToWorkPos => "BA030AZSBK30.02");
END_REGION

REGION Network 117: *************** Feedback to Unit ***************************
END_REGION

REGION Network 118: Determine StateComplete (SC) in Mode Production
   // Conditions for the Equipment Modules "stateComplete" feedback to the unit. This feedback is given when the task in for the respective state is complete.
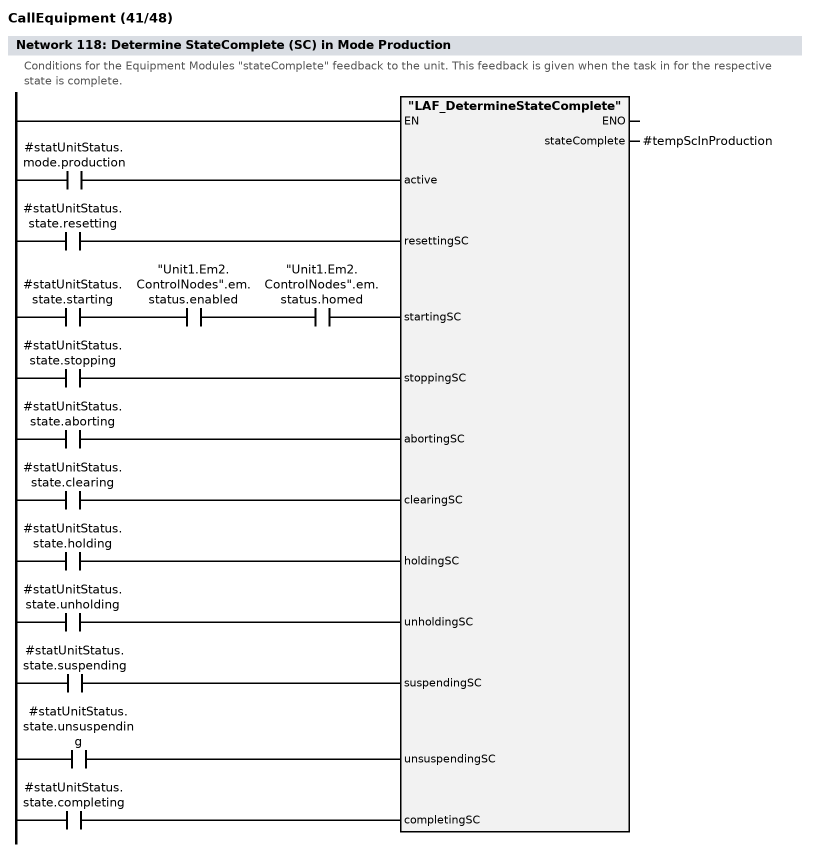
   RUNG wire#powerrail
      "LAF_DetermineStateComplete"(active := wire#w1, resettingSC := wire#w2, startingSC := wire#w3, stoppingSC := wire#w4, abortingSC := wire#w5, clearingSC := wire#w6, holdingSC := wire#w7, unholdingSC := wire#w8, suspendingSC := wire#w9, unsuspendingSC := wire#w10, completingSC := wire#w11, stateComplete => #tempScInProduction)
   END_RUNG
   RUNG wire#powerrail
      Contact( #statUnitStatus.mode.production )
   END_RUNG wire#w1
   RUNG wire#powerrail
      Contact( #statUnitStatus.state.resetting )
   END_RUNG wire#w2
   RUNG wire#powerrail
      Contact( #statUnitStatus.state.starting )
      Contact( "Unit1.Em2.ControlNodes".em.status.enabled )
      Contact( "Unit1.Em2.ControlNodes".em.status.homed )
   END_RUNG wire#w3
   RUNG wire#powerrail
      Contact( #statUnitStatus.state.stopping )
   END_RUNG wire#w4
   RUNG wire#powerrail
      Contact( #statUnitStatus.state.aborting )
   END_RUNG wire#w5
   RUNG wire#powerrail
      Contact( #statUnitStatus.state.clearing )
   END_RUNG wire#w6
   RUNG wire#powerrail
      Contact( #statUnitStatus.state.holding )
   END_RUNG wire#w7
   RUNG wire#powerrail
      Contact( #statUnitStatus.state.unholding )
   END_RUNG wire#w8
   RUNG wire#powerrail
      Contact( #statUnitStatus.state.suspending )
   END_RUNG wire#w9
   RUNG wire#powerrail
      Contact( #statUnitStatus.state.unsuspending )
   END_RUNG wire#w10
   RUNG wire#powerrail
      Contact( #statUnitStatus.state.completing )
   END_RUNG wire#w11
   // the same network as SCL:
   "LAF_DetermineStateComplete"(active := #statUnitStatus.mode.production,
                           resettingSC := #statUnitStatus.state.resetting,
                           startingSC := #statUnitStatus.state.starting AND "Unit1.Em2.ControlNodes".em.status.enabled AND "Unit1.Em2.ControlNodes".em.status.homed,
                           stoppingSC := #statUnitStatus.state.stopping,
                           abortingSC := #statUnitStatus.state.aborting,
                           clearingSC := #statUnitStatus.state.clearing,
                           holdingSC := #statUnitStatus.state.holding,
                           unholdingSC := #statUnitStatus.state.unholding,
                           suspendingSC := #statUnitStatus.state.suspending,
                           unsuspendingSC := #statUnitStatus.state.unsuspending,
                           completingSC := #statUnitStatus.state.completing,
                           stateComplete => #tempScInProduction);
END_REGION

REGION Network 119: Determine StateComplete (SC) in Mode Maintenance/Manual
   // Conditions for the Equipment Modules "stateComplete" feedback to the unit. This feedback is given when the task in for the respective state is complete.
